	IF State_HS = 0	THEN
		IF SI_MS[0].Event = INIT_CONTINUOUS THEN
			State_MS := 10;
		ELSE
			FSY_In   := FALSE;
			FSY_Out  := FALSE;
			BDef_In  := FALSE;
			BDef_Out := FALSE;
			TDef_In  := FALSE;
			TDef_Out := FALSE;
		END_IF
	END_IF

(*Select MainSail Position*)
10:
	IF END_MS OR Cnt_MS > 10.0 THEN
		State_MS := 0;

	(*1th*)
	ELSIF SI_MS[1].Event = INIT_CONTINUOUS THEN
		Cnt_MS      := 0.0;
		Selected_MS := 1;

		IF TABLE.aFSY [Selected_MS,Selected_HS] = 0
		OR TABLE.aBDef[Selected_MS,Selected_HS] = 0
		OR TABLE.aTDef[Selected_MS,Selected_HS] = 0
		THEN State_MS := 0;
		ELSE State_MS := 11;
		END_IF

	(*2th*)
	ELSIF SI_MS[2].Event = INIT_CONTINUOUS THEN
		Cnt_MS      := 0.0;
		Selected_MS := 2;

		IF TABLE.aFSY [Selected_MS,Selected_HS] = 0
		OR TABLE.aBDef[Selected_MS,Selected_HS] = 0
		OR TABLE.aTDef[Selected_MS,Selected_HS] = 0
		THEN State_MS := 0;
		ELSE State_MS := 12;
		END_IF

	(*3th*)
	ELSIF SI_MS[3].Event = INIT_CONTINUOUS THEN
		Cnt_MS      := 0.0;
		Selected_MS := 3;

		IF TABLE.aFSY [Selected_MS,Selected_HS] = 0
		OR TABLE.aBDef[Selected_MS,Selected_HS] = 0
		OR TABLE.aTDef[Selected_MS,Selected_HS] = 0
		THEN State_MS := 0;
		ELSE State_MS := 13;
		END_IF

	(*FULL*)
	ELSIF SI_MS[4].Event = INIT_CONTINUOUS THEN
		Cnt_MS      := 0.0;
		Selected_MS := 4;

		IF TABLE.aFSY [Selected_MS,Selected_HS] = 0
		OR TABLE.aBDef[Selected_MS,Selected_HS] = 0
		OR TABLE.aTDef[Selected_MS,Selected_HS] = 0
		THEN State_MS := 0;
		ELSE State_MS := 14;
		END_IF

	END_IF

(*Wait 5 Sec*)
11,12,13,14:
	IF END_MS THEN
		State_MS := 0;

	ELSIF Cnt_MS > 5.0 THEN
		Cnt_MS   := 0.0;

		FSY_Tgt := TABLE.aFSY [Selected_MS,Selected_HS];
		FSY_In  := NOT FSY_LS.Err AND FSY_LS.Pos > FSY_Tgt AND NOT FSY_P.AlMax;
		FSY_Out := NOT FSY_LS.Err AND FSY_LS.Pos < FSY_Tgt;

		State_MS := State_MS + 10;

	END_IF

(*Moving Forestay*)
21,22,23,24:
	IF END_MS OR Cnt_MS > 30.0 OR FSY_LS.Err THEN
		State_MS := 0;

	ELSIF FSY_In THEN
		IF FSY_P.AlMax THEN
			State_MS := 0;

		ELSIF FSY_LS.Pos <= FSY_Tgt THEN
			FSY_In   := FALSE;

			BDef_Tgt := TABLE.aBDef[Selected_MS,Selected_HS];
			BDef_In  := NOT BDef_LS.Err AND BDef_LS.Pos > BDef_Tgt AND NOT BDef_P.AlMax;
			BDef_Out := NOT BDef_LS.Err AND BDef_LS.Pos < BDef_Tgt;

			TDef_Tgt := TABLE.aTDef[Selected_MS,Selected_HS];
			TDef_In  := NOT TDef_LS.Err AND TDef_LS.Pos > TDef_Tgt AND NOT TDef_P.AlMax;
			TDef_Out := NOT TDef_LS.Err AND TDef_LS.Pos < TDef_Tgt;

			State_MS := State_MS + 10;

		END_IF

	ELSIF FSY_OUT THEN
		IF FSY_LS.Pos >= FSY_Tgt THEN
			FSY_Out  := FALSE;

			BDef_Tgt := TABLE.aBDef[Selected_MS,Selected_HS];
			BDef_In  := NOT BDef_LS.Err AND BDef_LS.Pos > BDef_Tgt AND NOT BDef_P.AlMax;
			BDef_Out := NOT BDef_LS.Err AND BDef_LS.Pos < BDef_Tgt;

			TDef_Tgt := TABLE.aTDef[Selected_MS,Selected_HS];
			TDef_In  := NOT TDef_LS.Err AND TDef_LS.Pos > TDef_Tgt AND NOT TDef_P.AlMax;
			TDef_Out := NOT TDef_LS.Err AND TDef_LS.Pos < TDef_Tgt;

			State_MS := State_MS + 10;

		END_IF

	ELSE
		State_MS := 0;

	END_IF

(*Moving Deflector*)
31,32,33,34:
	IF END_MS OR Cnt_MS > 30.0 OR BDef_LS.Err OR TDef_LS.Err THEN
		State_MS := 0;

	ELSE
		IF BDef_In THEN
			IF BDef_P.AlMax THEN
				State_MS := 0;
			ELSIF BDef_LS.Pos <= BDef_Tgt THEN
				BDef_In := FALSE;
			END_IF

		ELSIF BDef_Out THEN
			IF BDef_LS.Pos >= BDef_Tgt THEN
				BDef_Out := FALSE;
			END_IF
		END_IF

		IF TDef_In THEN
			IF TDef_P.AlMax THEN
				State_MS := 0;
			ELSIF TDef_LS.Pos <= TDef_Tgt THEN
				TDef_In := FALSE;
			END_IF

		ELSIF TDef_Out THEN
			IF TDef_LS.Pos >= TDef_Tgt THEN
				TDef_Out := FALSE;
			END_IF
		END_IF

		IF NOT BDef_In AND NOT BDef_OUT AND NOT TDef_In AND NOT TDef_Out THEN
			State_MS := 0;
		END_IF

	END_IF

END_CASE

(*HEAD SAIL*)
CASE State_HS OF
0:
	Cnt_HS := 0.0;

	IF State_MS = 0	THEN
		IF SI_HS[0].Event = INIT_CONTINUOUS THEN
			State_HS := 10;
		ELSE
			FSY_In   := FALSE;
			FSY_Out  := FALSE;
			BDef_In  := FALSE;
			BDef_Out := FALSE;
			TDef_In  := FALSE;
			TDef_Out := FALSE;
		END_IF
	END_IF

(*Select HeadSail*)
10:
	IF END_HS OR Cnt_HS > 10.0 THEN
		State_HS := 0;

	(*A3*)
	ELSIF SI_HS[1].Event = INIT_CONTINUOUS THEN
		Cnt_HS      := 0.0;
		Selected_HS := 1;

		IF TABLE.aFSY [Selected_MS,Selected_HS] = 0
		OR TABLE.aBDef[Selected_MS,Selected_HS] = 0
		OR TABLE.aTDef[Selected_MS,Selected_HS] = 0
		THEN State_HS := 0;
		ELSE State_HS := 11;
		END_IF

	(*F0*)
	ELSIF SI_HS[2].Event = INIT_CONTINUOUS THEN
		Cnt_HS      := 0.0;
		Selected_HS := 2;

		IF TABLE.aFSY [Selected_MS,Selected_HS] = 0
		OR TABLE.aBDef[Selected_MS,Selected_HS] = 0
		OR TABLE.aTDef[Selected_MS,Selected_HS] = 0
		THEN State_HS := 0;
		ELSE State_HS := 12;
		END_IF

	(*J2*)
	ELSIF SI_HS[3].Event = INIT_CONTINUOUS THEN
		Cnt_HS      := 0.0;
		Selected_HS := 3;

		IF TABLE.aFSY [Selected_MS,Selected_HS] = 0
		OR TABLE.aBDef[Selected_MS,Selected_HS] = 0
		OR TABLE.aTDef[Selected_MS,Selected_HS] = 0
		THEN State_HS := 0;
		ELSE State_HS := 13;
		END_IF

	(*J4*)
	ELSIF SI_HS[4].Event = INIT_CONTINUOUS THEN
		Cnt_HS      := 0.0;
		Selected_HS := 4;

		IF TABLE.aFSY [Selected_MS,Selected_HS] = 0
		OR TABLE.aBDef[Selected_MS,Selected_HS] = 0
		OR TABLE.aTDef[Selected_MS,Selected_HS] = 0
		THEN State_HS := 0;
		ELSE State_HS := 14;
		END_IF

	END_IF

(*Wait 5 Sec*)
11,12,13,14,15,16:
	IF END_HS THEN
		State_HS := 0;

	(*A3+J4*)
	ELSIF State_HS = 11 AND SI_HS[4].Event = INIT_CONTINUOUS THEN
		Cnt_HS      := 0.0;
		Selected_HS := 5;

		IF TABLE.aFSY [Selected_MS,Selected_HS] = 0
		OR TABLE.aBDef[Selected_MS,Selected_HS] = 0
		OR TABLE.aTDef[Selected_MS,Selected_HS] = 0
		THEN State_HS := 0;
		ELSE State_HS := 15;
		END_IF

	(*F0+J4*)
	ELSIF State_HS = 12 AND SI_HS[4].Event = INIT_CONTINUOUS THEN
		Cnt_HS      := 0.0;
		Selected_HS := 6;

		IF TABLE.aFSY [Selected_MS,Selected_HS] = 0
		OR TABLE.aBDef[Selected_MS,Selected_HS] = 0
		OR TABLE.aTDef[Selected_MS,Selected_HS] = 0
		THEN State_HS := 0;
		ELSE State_HS := 16;
		END_IF

	ELSIF Cnt_HS > 5.0 THEN
		Cnt_HS   := 0.0;

		FSY_Tgt := TABLE.aFSY [Selected_MS,Selected_HS];
		FSY_In  := NOT FSY_LS.Err AND FSY_LS.Pos > FSY_Tgt AND NOT FSY_P.AlMax;
		FSY_Out := NOT FSY_LS.Err AND FSY_LS.Pos < FSY_Tgt;

		State_HS := State_HS + 10;

	END_IF

(*Moving Forestay*)
21,22,23,24,25,26:
	IF END_HS OR Cnt_HS > 30.0 OR FSY_LS.Err THEN
		State_HS := 0;

	ELSIF FSY_In THEN
		IF FSY_P.AlMax THEN
			State_HS := 0;

		ELSIF FSY_LS.Pos <= FSY_Tgt THEN
			FSY_In   := FALSE;

			BDef_Tgt := TABLE.aBDef[Selected_MS,Selected_HS];
			BDef_In  := NOT BDef_LS.Err AND BDef_LS.Pos > BDef_Tgt AND NOT BDef_P.AlMax;
			BDef_Out := NOT BDef_LS.Err AND BDef_LS.Pos < BDef_Tgt;

			TDef_Tgt := TABLE.aTDef[Selected_MS,Selected_HS];
			TDef_In  := NOT TDef_LS.Err AND TDef_LS.Pos > TDef_Tgt AND NOT TDef_P.AlMax;
			TDef_Out := NOT TDef_LS.Err AND TDef_LS.Pos < TDef_Tgt;

			State_HS := State_HS + 10;

		END_IF

	ELSIF FSY_OUT THEN
		IF FSY_LS.Pos >= FSY_Tgt THEN
			FSY_Out  := FALSE;

			BDef_Tgt := TABLE.aBDef[Selected_MS,Selected_HS];
			BDef_In  := NOT BDef_LS.Err AND BDef_LS.Pos > BDef_Tgt AND NOT BDef_P.AlMax;
			BDef_Out := NOT BDef_LS.Err AND BDef_LS.Pos < BDef_Tgt;

			TDef_Tgt := TABLE.aTDef[Selected_MS,Selected_HS];
			TDef_In  := NOT TDef_LS.Err AND TDef_LS.Pos > TDef_Tgt AND NOT TDef_P.AlMax;
			TDef_Out := NOT TDef_LS.Err AND TDef_LS.Pos < TDef_Tgt;

			State_HS := State_HS + 10;

		END_IF

	ELSE
		State_HS := 0;

	END_IF

(*Moving Deflector*)
31,32,33,34,35,36:
	IF END_HS OR Cnt_HS > 30.0 OR BDef_LS.Err OR TDef_LS.Err THEN
		State_HS := 0;

	ELSE
		IF BDef_In THEN
			IF BDef_P.AlMax THEN
				State_HS := 0;
			ELSIF BDef_LS.Pos <= BDef_Tgt THEN
				BDef_In := FALSE;
			END_IF

		ELSIF BDef_Out THEN
			IF BDef_LS.Pos >= BDef_Tgt THEN
				BDef_Out := FALSE;
			END_IF
		END_IF

		IF TDef_In THEN
			IF TDef_P.AlMax THEN
				State_HS := 0;
			ELSIF TDef_LS.Pos <= TDef_Tgt THEN
				TDef_In := FALSE;
			END_IF

		ELSIF TDef_Out THEN
			IF TDef_LS.Pos >= TDef_Tgt THEN
				TDef_Out := FALSE;
			END_IF
		END_IF

		IF NOT BDef_In AND NOT BDef_OUT AND NOT TDef_In AND NOT TDef_Out THEN
			State_HS := 0;
		END_IF

	END_IF

END_CASE
END_FUNCTION_BLOCK

(* POU OUTPUTS, ST *)
PROGRAM OUTPUTS
VAR CONSTANT
	BUF_SIZE : WORD := 4095;
	MAX_PSX  : INT  := 1000; (*100*10*)
END_VAR
VAR
	PSX50 : FB_PSX_VALVE;
	PSX51 : FB_PSX_VALVE;
	PSX52 : FB_PSX_VALVE;
	PSX53 : FB_PSX_VALVE;
	PSX54 : FB_PSX_VALVE;
	PSX55 : FB_PSX_VALVE;
	PSX56 : FB_PSX_VALVE;
	PSX57 : FB_PSX_VALVE;
	PSX58 : FB_PSX_VALVE;
	PSX59 : FB_PSX_VALVE;

	PSX60 : FB_PSX_VALVE;
	PSX61 : FB_PSX_VALVE;
	PSX64 : FB_PSX_VALVE;

	PSX70 : FB_PSX_VALVE;
	PSX71 : FB_PSX_VALVE;
	PSX72 : FB_PSX_VALVE;
	PSX73 : FB_PSX_VALVE;
	PSX74 : FB_PSX_VALVE;

	tsTime    :TIMESTRUCT;
	sDate     :STRING;
	sLocal    :STRING;
	sDaySec   :STRING;


	SIMob      : FB_SMART_INPUT;
	SIDimmerUp : FB_SMART_INPUT;
	SIDimmerDw : FB_SMART_INPUT;

	wDimmerBackLight : WORD;
	byDimmerLedBar   : BYTE;
	byDimmerDeckLink : BYTE;
	byDimmerBLink    : BYTE;
	byDimmerState    : BYTE;

	(*Mob : BOOL;*)

	sValue : STRING;

	engCnt : REAL;

	(*UDP Stream*)
	fbUdpSend        : FB_UDP_SEND;
	fbSocketCloseAll : FB_SocketCloseAll;
    bCloseAll 	     : BOOL := TRUE;

	aBuffer : ARRAY[0..BUF_SIZE] OF BYTE;
	wBufPos : DWORD;

	i   : INT;
	chk : BYTE;
	(*Bobstay_Ignore : BOOL;*)


	fbResetCan1 : IOF_DeviceReset;
	fbResetCan2 : IOF_DeviceReset;
	fbResetCan3 : IOF_DeviceReset;
	fbResetCan4 : IOF_DeviceReset;
	fbResetCan5 : IOF_DeviceReset;

	ResetCan1 : BOOL;
	ResetCan2 : BOOL;
	ResetCan3 : BOOL;
	ResetCan4 : BOOL;
	ResetCan5 : BOOL;

	W_CAN_PWR : BOOL := TRUE;
	W_CAN_CNT : REAL := 20.0;

END_VAR
VAR PERSISTENT
	Dimmer_Panels   AT %Q*: WORD;
	Dimmer_LedBar   AT %Q*: WORD;
	Dimmer_DeckLink AT %Q*: WORD;

END_VAR
W_CAN_CNT := W_CAN_CNT + MAIN.Cycle_Time;
W_CAN_PWR := W_CAN_CNT > 20.0;

(*Node00-PLC*)
N0_DO1 := ALARMS.Buzzer;
(*N0_DO2 := Engine Stop*)
N0_DO3 := W_CAN_PWR;
N0_DO4 := ENGINE.Engine_ON;
(*N0_DO5 := Engine Ignition*)
(*N0_DO6 := Engine Start*)
N0_DO7 := KEY_PP1;
N0_DO8 := KEY_PP2;

N0_AO1 := REAL_TO_INT(THR_PP1 * 3276.7); (*0..10V*)
N0_AO2 := REAL_TO_INT(THR_PP2 * 3276.7); (*0..10V*)


IF NOT TANK.Enable OR ENGINE.Engine_STOP OR NOT MAIN.aSys_Enable[8] THEN

	IF engCnt > 5 THEN
		N0_DO2 := FALSE;
	ELSE
		engCnt := engCnt + MAIN.Cycle_Time;
	END_IF

ELSE
	N0_DO2 := TRUE;


END_IF

(***STERN Nodes***)
(*Node36/37 - TANK + GS + MF00 + PP *)
	N36_EVP3_CH1_2 := EVP001;
	N36_EVP2_CH1_4 := EVP002;

	N36_DO7_CH3_2 := EV1501;
	N36_DO6_CH3_4 := EV1502;

(*Node38 - LIGHT*)
	N38_DO3_CH1_2 := L_Red;
	N38_DO2_CH1_4 := L_Anchor;
	N38_DO1_CH2_2 := L_Steam;
	N38_DO0_CH2_4 := L_Deck;
	N38_DO7_CH3_2 := L_Nav;
(*	N38_DO6_CH3_4 := ;*)
	N38_DO5_CH4_2 := ENGINE.Engine_ON;
	N38_DO4_CH4_4 := ALARMS.Buzzer;

(*Node39 - MF10A - Keel*)
	N39_DO7_CH3_2 := EV1001;
	N39_DO6_CH3_4 := EV1003;
	N39_DO5_CH4_2 := EV1002;
	N39_DO4_CH4_4 := EV1004;

	N39_EVP3_CH1_2 := EVP1006;
	N39_EVP2_CH1_4 := EVP1008;
	N39_EVP1_CH2_2 := EVP1007;
	N39_EVP0_CH2_4 := EVP1009;

(*Node40 - MF10B - Keel*)
	N40_EVP3_CH1_2 := EVP1005.mA := REAL_TO_UINT(EVP1005.Bar * EVP1005.Cal_K + EVP1005.Cal_Off);
	N40_EVP2_CH1_4 := EVP1010.mA := REAL_TO_UINT(EVP1010.Bar * EVP1010.Cal_K + EVP1010.Cal_Off);

	N40_DO1_CH2_2 := EV1011;
	N40_DO0_CH2_4 := EV1012;

(*Node41 - MF05*)
	IF EVP513.Bar > 0 THEN
		N41_EVP3_CH1_2 := EVP513.mA := REAL_TO_UINT(EVP513.Bar * EVP513.Cal_K + EVP513.Cal_Off);
	ELSE
		N41_EVP3_CH1_2 := EVP513.mA := 0;
	END_IF

	N41_DO1_CH2_2 := EV501;
	N41_DO0_CH2_4 := EV502;
	N41_DO7_CH3_2 := EV503;
	N41_DO6_CH3_4 := EV504;
	N41_DO5_CH4_2 := EV505;
	N41_DO4_CH4_4 := EV506;
	N40_DO7_CH3_2 := EV507;
	N40_DO6_CH3_4 := EV508;

(*Node42 - MF01 EVC + PP*)
	N42_DO3_CH1_2 := EV107;
(*	N42_DO2_CH1_4 := *)
	N42_DO1_CH2_2 := EV105;
	N42_DO0_CH2_4 := EV106;
	N42_DO7_CH3_2 := EV103;
	N42_DO6_CH3_4 := EV104;
	N42_DO5_CH4_2 := EV101;
	N42_DO4_CH4_4 := EV102;

(*Node43 - MF03A*)
	N43_DO3_CH1_2 := EV311;
	N43_DO2_CH1_4 := EV312;
	N43_DO1_CH2_2 := EV309;
	N43_DO0_CH2_4 := EV310;
	N43_DO7_CH3_2 := EV307;
	N43_DO6_CH3_4 := EV308;

(*Node44 - MF03A*)
	IF EVP313.Bar > 0 THEN
		N44_EVP3_CH1_2 := EVP313.mA := REAL_TO_UINT(EVP313.Bar * EVP313.Cal_K + EVP313.Cal_Off);
	ELSE
		N44_EVP3_CH1_2 := EVP313.mA := 0;
	END_IF

	N44_DO1_CH2_2 := EV301;
	N44_DO0_CH2_4 := EV302;
	N44_DO7_CH3_2 := EV303;
	N44_DO6_CH3_4 := EV304;
	N44_DO5_CH4_2 := EV305;
	N44_DO4_CH4_4 := EV306;

(*Node48 - DGB Seal*)
	N48_DO3_CH1_2 := EV_SealP_V;
	N48_DO2_CH1_4 := EV_SealP_P;
	N48_DO1_CH2_2 := EV_SealS_V;
	N48_DO0_CH2_4 := EV_SealS_P;

(***STERN Nodes***)
(*Node20 - MF06*)
	N20_DO3_CH1_2 := EV601;
	N20_DO2_CH1_4 := EV602;
	N20_DO1_CH2_2 := EV603;
	N20_DO0_CH2_4 := EV604;
	N20_DO7_CH3_2 := EV605;
	N20_DO6_CH3_4 := EV606;
	N20_DO5_CH4_2 := EV607;
	N20_DO4_CH4_4 := EV608;

(*Node21/22 - MF07 - MF10*)
	IF EVP709.Bar > 0 THEN
		N21_EVP3_CH1_2 := EVP709.mA := REAL_TO_UINT(EVP709.Bar * EVP709.Cal_K + EVP709.Cal_Off);
	ELSE
		N21_EVP3_CH1_2 := EVP709.mA := 0;
	END_IF

	N21_DO1_CH2_2 := EV701;
	N21_DO0_CH2_4 := EV702;
	N21_DO5_CH4_2 := EV703;
	N21_DO4_CH4_4 := EV704;

	N22_DO3_CH1_2 := EV709;
	N22_DO2_CH1_4 := EV710;
	N22_DO1_CH2_2 := EV707;
	N22_DO0_CH2_4 := EV708;
	N22_DO7_CH3_2 := EV705;
	N22_DO6_CH3_4 := EV706;

(*Node23 - MF08*)
	N23_DO3_CH1_2 := EV803;
	N23_DO2_CH1_4 := EV804;
	N23_DO1_CH2_2 := EV801;
	N23_DO0_CH2_4 := EV802;

(*Node26 - MF25*)
	N26_DO3_CH1_2 := EV2502;
	N26_DO2_CH1_4 := EV2504;
	N26_DO1_CH2_2 := EV2501;
	N26_DO0_CH2_4 := EV2503;
	N26_DO7_CH3_2 := EV2506;
	N26_DO6_CH3_4 := EV2508;
	N26_DO5_CH4_2 := EV2505;
	N26_DO4_CH4_4 := EV2507;

(*Node27 - MF22*)
	N27_DO3_CH1_2 := EV2211;
	N27_DO2_CH1_4 := EV2209;
	N27_DO1_CH2_2 := EV2207;
	N27_DO0_CH2_4 := EV2205;
	N27_DO7_CH3_2 := EV2203;
	N27_DO6_CH3_4 := EV2201;

(*Node28 - MF21*)
	N28_DO3_CH1_2 := EV2111;
	N28_DO2_CH1_4 := EV2109;
	N28_DO1_CH2_2 := EV2107;
	N28_DO0_CH2_4 := EV2105;
	N28_DO7_CH3_2 := EV2103;
	N28_DO6_CH3_4 := EV2101;

(*Node29 - MF24*)
	N29_DO3_CH1_2 := EV2411;
	N29_DO2_CH1_4 := EV2409;
	N29_DO1_CH2_2 := EV2407;
	N29_DO0_CH2_4 := EV2405;
	N29_DO7_CH3_2 := EV2403;
	N29_DO6_CH3_4 := EV2401;

(*Node30 - MF23*)
	N30_DO3_CH1_2 := EV2311;
	N30_DO2_CH1_4 := EV2309;
	N30_DO1_CH2_2 := EV2307;
	N30_DO0_CH2_4 := EV2305;
	N30_DO7_CH3_2 := EV2303;
	N30_DO6_CH3_4 := EV2301;

(*Node31 - MF20*)
	N31_DO3_CH1_2 := EV2011;
	N31_DO2_CH1_4 := EV2009;
	N31_DO1_CH2_2 := EV2007;
	N31_DO0_CH2_4 := EV2005;
	N31_DO7_CH3_2 := EV2003;
	N31_DO6_CH3_4 := EV2001;

(*Node32 - MF19*)
	N32_DO3_CH1_2 := EV1911;
	N32_DO2_CH1_4 := EV1909;
	N32_DO1_CH2_2 := EV1907;
	N32_DO0_CH2_4 := EV1905;
	N32_DO7_CH3_2 := EV1903;
	N32_DO6_CH3_4 := EV1901;

(*Node33 - MF13 - Traveller*)
	N33_DO3_CH1_2 := EV1302;
	N33_DO2_CH1_4 := EV1301;
	N33_DO1_CH2_2 := EV1303;

(*Node35 - MF09 - Traveller*)
(*	IF EVP905.Bar > 0 THEN
		N35_EVP3_CH1_2 := EVP905.mA := REAL_TO_UINT(EVP905.Bar * EVP905.Cal_K + EVP905.Cal_Off);
	ELSE
		N35_EVP3_CH1_2 := EVP905.mA := 0;
	END_IF*)

	N35_DO3_CH1_2 := EV905;
	N35_DO2_CH1_4 := EV906;
	N35_DO1_CH2_2 := EV901;
	N35_DO0_CH2_4 := EV902;
	N35_DO7_CH3_2 := EV903;
	N35_DO6_CH3_4 := EV904;
	N35_DO5_CH4_2 := EV907;
	N35_DO4_CH4_4 := EV908;

(*Node47 - MF11*)
	N47_DO1_CH2_2 := EV1101;

(*Node50/59*)
	IF NOT ENGINE.Engine_ON THEN
		IF    EVP402_3 > 0 THEN EVP402_3 :=  MAX_PSX;
		ELSIF EVP402_3 < 0 THEN EVP402_3 := -MAX_PSX;
		END_IF
		IF    EVP404_5 > 0 THEN EVP404_5 :=  MAX_PSX;
		ELSIF EVP404_5 < 0 THEN EVP404_5 := -MAX_PSX;
		END_IF
		IF    EVP406_7 > 0 THEN EVP406_7 :=  MAX_PSX;
		ELSIF EVP406_7 < 0 THEN EVP406_7 := -MAX_PSX;
		END_IF

		IF    EVP1202_3 > 0 THEN EVP1202_3 :=  MAX_PSX;
		ELSIF EVP1202_3 < 0 THEN EVP1202_3 := -MAX_PSX;
		END_IF
		IF    EVP1204_5 > 0 THEN EVP1204_5 :=  MAX_PSX;
		ELSIF EVP1204_5 < 0 THEN EVP1204_5 := -MAX_PSX;
		END_IF
		IF    EVP1206_7 > 0 THEN EVP1206_7 :=  MAX_PSX;
		ELSIF EVP1206_7 < 0 THEN EVP1206_7 := -MAX_PSX;
		END_IF
		IF    EVP1208_9 > 0 THEN EVP1208_9 :=  MAX_PSX;
		ELSIF EVP1208_9 < 0 THEN EVP1208_9 := -MAX_PSX;
		END_IF
		IF    EVP1210_1 > 0 THEN EVP1210_1 :=  MAX_PSX;
		ELSIF EVP1210_1 < 0 THEN EVP1210_1 := -MAX_PSX;
		END_IF
		IF    EVP1212_3 > 0 THEN EVP1212_3 :=  MAX_PSX;
		ELSIF EVP1212_3 < 0 THEN EVP1212_3 := -MAX_PSX;
		END_IF
		IF    EVP1214_5 > 0 THEN EVP1214_5 :=  MAX_PSX;
		ELSIF EVP1214_5 < 0 THEN EVP1214_5 := -MAX_PSX;
		END_IF
		(*IF  EVP1216_7 > 0 THEN EVP1216_7 :=  MAX_PSX; (*Board. Proper value when not Engine.*)
		ELSIF EVP1216_7 < 0 THEN EVP1216_7 := -MAX_PSX;
		END_IF
		IF    EVP1218_9 > 0 THEN EVP1218_9 :=  MAX_PSX;
		ELSIF EVP1218_9 < 0 THEN EVP1218_9 := -MAX_PSX;
		END_IF*)
		(*IF  EVP1220_1 > 0 THEN EVP1220_1 :=  MAX_PSX; (*Keel Fill. Not Without Engine.*)
		ELSIF EVP1220_1 < 0 THEN EVP1220_1 :=  0;
		END_IF*)

		IF    EVP1602_3 > 0 THEN EVP1602_3 :=  MAX_PSX;
		ELSIF EVP1602_3 < 0 THEN EVP1602_3 := -MAX_PSX;
		END_IF
		IF    EVP1604_5 > 0 THEN EVP1604_5 :=  MAX_PSX;
		ELSIF EVP1604_5 < 0 THEN EVP1604_5 := -MAX_PSX;
		END_IF
		IF    EVP1606_7 > 0 THEN EVP1606_7 :=  MAX_PSX;
		ELSIF EVP1606_7 < 0 THEN EVP1606_7 := -MAX_PSX;
		END_IF
		IF    EVP1608_9 > 0 THEN EVP1608_9 :=  MAX_PSX;
		ELSIF EVP1608_9 < 0 THEN EVP1608_9 := -MAX_PSX;
		END_IF
		IF    EVP1610_1 > 0 THEN EVP1610_1 :=  MAX_PSX;
		ELSIF EVP1610_1 < 0 THEN EVP1610_1 := -MAX_PSX;
		END_IF

	END_IF

	PSX50( SP:= EVP1202_3, IN:= N50_IN, OUT:= N50_OUT );
	PSX51( SP:= EVP1204_5, IN:= N51_IN, OUT:= N51_OUT );
	PSX52( SP:= EVP1206_7, IN:= N52_IN, OUT:= N52_OUT );
	PSX53( SP:= EVP1208_9, IN:= N53_IN, OUT:= N53_OUT );
	PSX54( SP:= EVP1210_1, IN:= N54_IN, OUT:= N54_OUT );
	PSX55( SP:= EVP1212_3, IN:= N55_IN, OUT:= N55_OUT );
	PSX56( SP:= EVP1214_5, IN:= N56_IN, OUT:= N56_OUT );
	PSX57( SP:= EVP1216_7, IN:= N57_IN, OUT:= N57_OUT );
	PSX58( SP:= EVP1218_9, IN:= N58_IN, OUT:= N58_OUT );
	PSX59( SP:= EVP1220_1, IN:= N59_IN, OUT:= N59_OUT );

	PSX60( SP:= EVP402_3, IN:= N60_IN, OUT:= N60_OUT );
	PSX61( SP:= EVP404_5, IN:= N61_IN, OUT:= N61_OUT );
	PSX64( SP:= EVP406_7, IN:= N64_IN, OUT:= N64_OUT );

	PSX70( SP:= EVP1602_3, IN:= N70_IN, OUT:= N70_OUT );
	PSX71( SP:= EVP1604_5, IN:= N71_IN, OUT:= N71_OUT );
	PSX72( SP:= EVP1606_7, IN:= N72_IN, OUT:= N72_OUT );
	PSX73( SP:= EVP1608_9, IN:= N73_IN, OUT:= N73_OUT );
	PSX74( SP:= EVP1610_1, IN:= N74_IN, OUT:= N74_OUT );

(*-------------------*)
(*-- Panel Buttons --*)
(*-------------------*)
SIDimmerUp( T_Cont:= T#0ms, T_DClk:= T#0ms);
SIDimmerDw(In:= N103_IN.5, T_Cont:= T#0ms, T_DClk:= T#0ms);

IF SIDimmerUp.Event = INIT_CONTINUOUS
OR SIDimmerDw.Event = INIT_CONTINUOUS
THEN

	IF byDimmerState = 2
	THEN byDimmerState := 0;
	ELSE byDimmerState := byDimmerState + 1;
	END_IF

END_IF

CASE byDimmerState OF
0:
	wDimmerBackLight := 100;
	byDimmerLedBar   := 16#9F; (*16#80 + 16#1F*)
	byDimmerDeckLink := 16#07;
	byDimmerBLink    := 16#3F;

1:
	wDimmerBackLight := Dimmer_Panels;
	byDimmerLedBar   := REAL_TO_USINT(Dimmer_LedBar   * 0.31) + 16#80;
	byDimmerDeckLink := REAL_TO_USINT(Dimmer_DEckLink * 0.07);
	byDimmerBLink    := REAL_TO_USINT(Dimmer_Panels   * 0.63);

2:
	wDimmerBackLight := 100;
	byDimmerLedBar   := 16#9F; (*16#80 + 16#1F*)
	byDimmerDeckLink := 16#07;
	byDimmerBLink    := 16#3F;

END_CASE

IF byDimmerState > 0 AND MAIN.aSys_Enable[2] AND wDimmerBackLight > 0 THEN
	N102_OUT := 16#FFFF;
	N103_OUT := 16#FFFF;
	N104_OUT := 16#FFFF;
	N105_OUT := 16#FFFF;
	N106_OUT := 16#FFFF;
	N107_OUT := 16#FFFF;
	N108_OUT := 16#FFE0;
	N109_OUT := 16#FFE0;
	N110_OUT := 16#FFFF;
	N111_OUT := 16#FFFF;
	N112_OUT := 16#FFFF;
	N113_OUT := 16#FFFF;
	N114_OUT := 16#FFFF;
	N115_OUT := 16#FFFF;
	N116_OUT := 16#FFFF;
	N117_OUT := 16#FFFF;
	N118_OUT := 16#FFFF;
	N119_OUT := 16#FFFF;

	N120_LED_R := 16#0000;
	N120_LED_G := 16#03DE;
	N120_LED_B := 16#0021;
	N121_LED_R := 16#00FF;
	N121_LED_G := 16#0000;
	N121_LED_B := 16#0000;

ELSE
	N102_OUT := 0;
	N103_OUT := 0;
	N104_OUT := 0;
	N105_OUT := 0;
	N106_OUT := 0;
	N107_OUT := 0;
	N108_OUT := 0;
	N109_OUT := 0;
	N110_OUT := 0;
	N111_OUT := 0;
	N112_OUT := 0;
	N113_OUT := 0;
	N114_OUT := 0;
	N115_OUT := 0;
	N116_OUT := 0;
	N117_OUT := 0;
	N118_OUT := 0;
	N119_OUT := 0;

	N120_LED_R := 0;
	N120_LED_G := 0;
	N120_LED_B := 0;
	N121_LED_R := 0;
	N121_LED_G := 0;
	N121_LED_B := 0;
END_IF

IF wDimmerBackLight = 0 THEN wDimmerBackLight := 1; END_IF

N102_DIMMER := wDimmerBackLight;
N103_DIMMER := wDimmerBackLight;
N104_DIMMER := wDimmerBackLight;
N105_DIMMER := wDimmerBackLight;
N106_DIMMER := wDimmerBackLight;
N107_DIMMER := wDimmerBackLight;
N108_DIMMER := wDimmerBackLight;
N109_DIMMER := wDimmerBackLight;
N110_DIMMER := wDimmerBackLight;
N111_DIMMER := wDimmerBackLight;
N112_DIMMER := wDimmerBackLight;
N113_DIMMER := wDimmerBackLight;
N114_DIMMER := wDimmerBackLight;
N115_DIMMER := wDimmerBackLight;
N116_DIMMER := wDimmerBackLight;
N117_DIMMER := wDimmerBackLight;
N118_DIMMER := wDimmerBackLight;
N119_DIMMER := wDimmerBackLight;

N120_LED_Bright := byDimmerBLink;
N121_LED_Bright := byDimmerBLink;

N102_BTIME := 10;
N103_BTIME := 10;
N104_BTIME := 10;
N105_BTIME := 10;
IF MAIN.fbWB.Pause THEN
	N106_BTIME := 100;
	N107_BTIME := 100;
ELSE
	N106_BTIME := 10;
	N107_BTIME := 10;
END_IF
N108_BTIME := 10;
N109_BTIME := 10;
N110_BTIME := 10;
N111_BTIME := 10;
N112_BTIME := 10;
N113_BTIME := 10;
N114_BTIME := 10;
N115_BTIME := 10;
N116_BTIME := 10;
N117_BTIME := 10;
N118_BTIME := 10;
N119_BTIME := 10;

(*FRO TACK*)
N102_BLINK.2 := MAIN.fbSE301.OUT_CylIn;
N102_BLINK.3 := MAIN.fbSE301.OUT_CylOut;
N113_BLINK.3 := MAIN.fbSE301.OUT_CylIn;
N113_BLINK.2 := MAIN.fbSE301.OUT_CylOut;
(*A3 TACK*)
N102_BLINK.4 := MAIN.fbSE303.OUT_CylIn;
N102_BLINK.5 := MAIN.fbSE303.OUT_CylOut;
N113_BLINK.5 := MAIN.fbSE303.OUT_CylIn;
N113_BLINK.4 := MAIN.fbSE303.OUT_CylOut;
(*J5*)
N118_BLINK.6 := MAIN.fbSE305.OUT_CylIn;
N118_BLINK.7 := MAIN.fbSE305.OUT_CylOut;
N119_BLINK.7 := MAIN.fbSE305.OUT_CylIn;
N119_BLINK.6 := MAIN.fbSE305.OUT_CylOut;
(*J4*)
N118_BLINK.8 := MAIN.fbSE307.OUT_CylIn;
N118_BLINK.9 := MAIN.fbSE307.OUT_CylOut;
N119_BLINK.9 := MAIN.fbSE307.OUT_CylIn;
N119_BLINK.8 := MAIN.fbSE307.OUT_CylOut;
(*FORESTAY*)
N104_BLINK.1 := MAIN.fbSE309.OUT_CylIn;
N104_BLINK.0 := MAIN.fbSE309.OUT_CylOut;
N105_BLINK.0 := MAIN.fbSE309.OUT_CylIn;
N105_BLINK.1 := MAIN.fbSE309.OUT_CylOut;
(*J2*)
N114_BLINK.4 := MAIN.fbSE311.OUT_CylIn;
N114_BLINK.5 := MAIN.fbSE311.OUT_CylOut;
N115_BLINK.5 := MAIN.fbSE311.OUT_CylIn;
N115_BLINK.4 := MAIN.fbSE311.OUT_CylOut;

(*JIB INOUT*)
N114_BLINK.2 := MAIN.fbSE501.OUT_CylIn;
N114_BLINK.3 := MAIN.fbSE501.OUT_CylOut;
N115_BLINK.3 := MAIN.fbSE501.OUT_CylIn;
N115_BLINK.2 := MAIN.fbSE501.OUT_CylOut;
(*JIB UPDW*)
N114_BLINK.0 := MAIN.fbSE503.OUT_CylIn;
N114_BLINK.1 := MAIN.fbSE503.OUT_CylOut;
N115_BLINK.1 := MAIN.fbSE503.OUT_CylIn;
N115_BLINK.0 := MAIN.fbSE503.OUT_CylOut;
(*VANG*)
N116_BLINK.2 := MAIN.fbSE505.OUT_CylIn;
N116_BLINK.3 := MAIN.fbSE505.OUT_CylOut;
N117_BLINK.3 := MAIN.fbSE505.OUT_CylIn;
N117_BLINK.2 := MAIN.fbSE505.OUT_CylOut;

(*PROP UPDW*)
N112_BLINK.3 := MAIN.fbDE601.OUT_EV3;
N112_BLINK.2 := MAIN.fbDE601.OUT_EV1;
(*TRIM TAB*)
N104_BLINK.3 := MAIN.fbDE605.OUT_EV3;
N104_BLINK.2 := MAIN.fbDE605.OUT_EV1;
N105_BLINK.3 := MAIN.fbDE605.OUT_EV3;
N105_BLINK.2 := MAIN.fbDE605.OUT_EV1;

(*INNER STAYSAIL*)
N102_BLINK.0 := MAIN.fbSE701.OUT_CylIn;
N102_BLINK.1 := MAIN.fbSE701.OUT_CylOut;
N113_BLINK.1 := MAIN.fbSE701.OUT_CylIn;
N113_BLINK.0 := MAIN.fbSE701.OUT_CylOut;
(*MAIN OUTHAUL*)
N116_BLINK.8 := MAIN.fbSE703.OUT_CylIn;
N116_BLINK.9 := MAIN.fbSE703.OUT_CylOut;
N117_BLINK.9 := MAIN.fbSE703.OUT_CylIn;
N117_BLINK.8 := MAIN.fbSE703.OUT_CylOut;
(*MAIN CUNN*)
N116_BLINK.6 := MAIN.fbSE705.OUT_CylIn;
N116_BLINK.7 := MAIN.fbSE705.OUT_CylOut;
N117_BLINK.7 := MAIN.fbSE705.OUT_CylIn;
N117_BLINK.6 := MAIN.fbSE705.OUT_CylOut;
(*BOTTOM DEF*)
N118_BLINK.2 := MAIN.fbSE707.OUT_CylIn;
N118_BLINK.3 := MAIN.fbSE707.OUT_CylOut;
N119_BLINK.3 := MAIN.fbSE707.OUT_CylIn;
N119_BLINK.2 := MAIN.fbSE707.OUT_CylOut;
(*BOTTOM DEF*)
N118_BLINK.4 := MAIN.fbSE709.OUT_CylIn;
N118_BLINK.5 := MAIN.fbSE709.OUT_CylOut;
N119_BLINK.5 := MAIN.fbSE709.OUT_CylIn;
N119_BLINK.4 := MAIN.fbSE709.OUT_CylOut;

(*BACKSTAY PORT*)
N104_BLINK.7 := MAIN.fbBSY.OUT_P_In;
N104_BLINK.6 := MAIN.fbBSY.OUT_P_Out;
N118_BLINK.0 := MAIN.fbBSY.OUT_P_In;
N118_BLINK.1 := MAIN.fbBSY.OUT_P_Out;
(*BACKSTAY STBD*)
N105_BLINK.6 := MAIN.fbBSY.OUT_S_In;
N105_BLINK.7 := MAIN.fbBSY.OUT_S_Out;
N119_BLINK.1 := MAIN.fbBSY.OUT_S_In;
N119_BLINK.0 := MAIN.fbBSY.OUT_S_Out;
(*BACKSTAY TACK*)
(*N104_BLINK.5 :=;*)
(*N105_BLINK.4 :=;*)

(*TRAVELLER*)
N116_BLINK.3 := MAIN.fbTraveller.Move_A;
N116_BLINK.2 := MAIN.fbTraveller.Move_B;
(*N116_BLINK.1 := ;*)
N116_BLINK.0 := MAIN.fbTraveller.OUT_EVAB;

N117_BLINK.3 := MAIN.fbTraveller.Move_A;
N117_BLINK.2 := MAIN.fbTraveller.Move_B;
(*N117_BLINK.0 := ;*)
N117_BLINK.1 := MAIN.fbTraveller.OUT_EVAB;

(*KEEL*)
N110_BLINK.0 := MAIN.fbKeel.MOVING_O;
N110_BLINK.4 := MAIN.fbKeel.MOVING_I;
N110_BLINK.3 := MAIN.fbKeel.MOVING_C;
N110_BLINK.2 := MAIN.fbKeel.MOVING_F;
N110_BLINK.5 := MAIN.fbKeel.MOVING_T;

N111_BLINK.0 := MAIN.fbKeel.MOVING_O;
N111_BLINK.4 := MAIN.fbKeel.MOVING_I;
N111_BLINK.3 := MAIN.fbKeel.MOVING_C;
N111_BLINK.2 := MAIN.fbKeel.MOVING_F;
N111_BLINK.5 := MAIN.fbKeel.MOVING_T;

(*N108_BLINK.0 := MAIN.fbKeel.MOVING_O;
N108_BLINK.4 := MAIN.fbKeel.MOVING_I;
N108_BLINK.3 := MAIN.fbKeel.MOVING_C;
N108_BLINK.2 := MAIN.fbKeel.MOVING_F;

N109_BLINK.0 := MAIN.fbKeel.MOVING_O;
N109_BLINK.4 := MAIN.fbKeel.MOVING_I;
N109_BLINK.3 := MAIN.fbKeel.MOVING_C;
N109_BLINK.2 := MAIN.fbKeel.MOVING_F;*) (*Now Mast setup*)

(*WINCHES*)
N117_BLINK.1 := INPUTS.Override_ON;
N105_BLINK.4 := INPUTS.RemPort_ON;
N104_BLINK.5 := INPUTS.RemStbd_ON;

(*MAINSAIL*)
CASE MAIN.fbMastSetup.State_MS OF
0: 	N109_BLINK.0 := N109_BLINK.4 := N109_BLINK.3 := N109_BLINK.2 := FALSE;

10:	N109_BLINK.0 := N109_BLINK.4 := N109_BLINK.3 := N109_BLINK.2 := TRUE;

11: N109_OUT.2   := TRUE;
	N109_BLINK.0 := N109_BLINK.4 := N109_BLINK.3 := N109_BLINK.2 := FALSE;

12: N109_OUT.4   := TRUE;
	N109_BLINK.0 := N109_BLINK.4 := N109_BLINK.3 := N109_BLINK.2 := FALSE;

13: N109_OUT.3   := TRUE;
	N109_BLINK.0 := N109_BLINK.4 := N109_BLINK.3 := N109_BLINK.2 := FALSE;

14: N109_OUT.0   := TRUE;
	N109_BLINK.0 := N109_BLINK.4 := N109_BLINK.3 := N109_BLINK.2 := FALSE;

21,31:
	N109_BLINK.2 := TRUE;
	N109_BLINK.0 := N109_BLINK.4 := N109_BLINK.3 := FALSE;

22,32:
	N109_BLINK.4 := TRUE;
	N109_BLINK.0 := N109_BLINK.3 := N109_BLINK.2 := FALSE;

23,33:
	N109_BLINK.3 := TRUE;
	N109_BLINK.0 := N109_BLINK.4 := N109_BLINK.2 := FALSE;

24,34:
	N109_BLINK.0 := TRUE;
	N109_BLINK.4 := N109_BLINK.3 := N109_BLINK.2 := FALSE;

END_CASE

(*HEADSAIL*)
CASE MAIN.fbMastSetup.State_HS OF
0: 	N108_BLINK.0 := N108_BLINK.4 := N108_BLINK.3 := N108_BLINK.2 := FALSE;

10: N108_BLINK.0 := N108_BLINK.4 := N108_BLINK.3 := N108_BLINK.2 := TRUE;

11:	N108_OUT.0   := TRUE;
	N108_BLINK.0 := N108_BLINK.4 := N108_BLINK.3 := N108_BLINK.2 := FALSE;

12:	N108_OUT.4   := TRUE;
	N108_BLINK.0 := N108_BLINK.4 := N108_BLINK.3 := N108_BLINK.2 := FALSE;

13:	N108_OUT.2   := TRUE;
	N108_BLINK.0 := N108_BLINK.4 := N108_BLINK.3 := N108_BLINK.2 := FALSE;

14:	N108_OUT.3   := TRUE;
	N108_BLINK.0 := N108_BLINK.4 := N108_BLINK.3 := N108_BLINK.2 := FALSE;

15:	N108_OUT.0   := N108_OUT.3   := TRUE;
	N108_BLINK.0 := N108_BLINK.4 := N108_BLINK.3 := N108_BLINK.2 := FALSE;

16:	N108_OUT.4   := N108_OUT.3   := TRUE;
	N108_BLINK.0 := N108_BLINK.4 := N108_BLINK.3 := N108_BLINK.2 := FALSE;

21,31:
	N108_BLINK.0 := TRUE;
	N108_BLINK.4 := N108_BLINK.3 := N108_BLINK.2 := FALSE;

22,32:
	N108_BLINK.4 := TRUE;
	N108_BLINK.0 := N108_BLINK.3 := N108_BLINK.2 := FALSE;

23,33:
	N108_BLINK.2 := TRUE;
	N108_BLINK.0 := N108_BLINK.4 := N108_BLINK.3 := FALSE;

24,34:
	N108_BLINK.3 := TRUE;
	N108_BLINK.0 := N108_BLINK.4 := N108_BLINK.2 := FALSE;

25,35:
	N108_BLINK.0 := N108_BLINK.3 := TRUE;
	N108_BLINK.4 := N108_BLINK.2 := FALSE;

26,36:
	N108_BLINK.4 := N108_BLINK.3 := TRUE;
	N108_BLINK.0 := N108_BLINK.2 := FALSE;

END_CASE

(*BOARD*)
N108_BLINK.6 := MAIN.fbBoard.MOVING_P;
N108_BLINK.7 := MAIN.fbBoard.MOVING_S;
N108_BLINK.5 := MAIN.fbBoard.MOVING_C;

N109_BLINK.6 := MAIN.fbBoard.MOVING_P;
N109_BLINK.7 := MAIN.fbBoard.MOVING_S;
N109_BLINK.5 := MAIN.fbBoard.MOVING_C;

(*BOW THR*)
N112_BLINK.4 := MAIN.fbBowThrUpDw.OUT_1;
N112_BLINK.5 := MAIN.fbBowThrUpDw.OUT_2;

(*Water Ballast*)
N106_BLINK.0 := N107_BLINK.0 := MAIN.fbWB.OUT_P_Fwd;
N106_BLINK.1 := N107_BLINK.1 := MAIN.fbWB.OUT_S_Fwd;
N106_BLINK.2 := N107_BLINK.2 := MAIN.fbWB.OUT_P_Aft;
N106_BLINK.3 := N107_BLINK.3 := MAIN.fbWB.OUT_S_Aft;
N106_BLINK.4 := N107_BLINK.4 := MAIN.fbWB.OUT_Fill;
N106_BLINK.5 := N107_BLINK.5 := MAIN.fbWB.OUT_Dump;
N106_BLINK.7 := N107_BLINK.7 := MAIN.fbWB.OUT_Stop;
N106_BLINK.8 := N107_BLINK.8 := MAIN.fbWB.OUT_12;
N106_BLINK.9 := N107_BLINK.9 := MAIN.fbWB.OUT_Move;

N120_BLINK_B.0 := MAIN.fbW1206.Out_1;
N120_BLINK_G.1 := MAIN.fbW1204.Out_1;
N120_BLINK_G.2 := MAIN.fbW1604.Out_1;
N120_BLINK_G.3 := MAIN.fbW1202.Out_1;
N120_BLINK_G.4 := MAIN.fbW1602.Out_1;
N120_BLINK_B.5 := MAIN.fbW1206.Out_2;
N120_BLINK_G.6 := MAIN.fbW1204.Out_2;
N120_BLINK_G.7 := MAIN.fbW1604.Out_2;
N120_BLINK_G.8 := MAIN.fbW1202.Out_2;
N120_BLINK_G.9 := MAIN.fbW1602.Out_2;

N121_BLINK_R.0 := MAIN.fbW1208.Out_1;
N121_BLINK_R.1 := MAIN.fbW1210.Out_1;
N121_BLINK_R.2 := MAIN.fbW1212.Out_1;
N121_BLINK_R.3 := MAIN.fbW1214.Out_1;
N121_BLINK_R.4 := MAIN.fbW1208.Out_2;
N121_BLINK_R.5 := MAIN.fbW1210.Out_2;
N121_BLINK_R.6 := MAIN.fbW1212.Out_2;
N121_BLINK_R.7 := MAIN.fbW1214.Out_2;

(*CLM8*)
CLM8_LED1.7 := TOFARO.rBar1 >= 100;
CLM8_LED1.6 := TOFARO.rBar1 >= 95;
CLM8_LED1.5 := TOFARO.rBar1 >= 90;
CLM8_LED1.4 := TOFARO.rBar1 >= 85;
CLM8_LED1.3 := TOFARO.rBar1 >= 68;
CLM8_LED1.2 := TOFARO.rBar1 >= 51;
CLM8_LED1.1 := TOFARO.rBar1 >= 34;
CLM8_LED1.0 := TOFARO.rBar1 >= 17;

CLM8_LED2.0 := TOFARO.rBar2 >= 100;
CLM8_LED2.1 := TOFARO.rBar2 >= 95;
CLM8_LED2.2 := TOFARO.rBar2 >= 90;
CLM8_LED2.3 := TOFARO.rBar2 >= 85;
CLM8_LED2.4 := TOFARO.rBar2 >= 68;
CLM8_LED2.5 := TOFARO.rBar2 >= 51;
CLM8_LED2.6 := TOFARO.rBar2 >= 34;
CLM8_LED2.7 := TOFARO.rBar2 >= 17;

IF TOFARO.rBar1 >= 105 THEN
				   (*7888____5556667722333444____1112*)
				   (*RBGR____BGRBGRBGGRBGRBGR____BGRB*)
	CLM8_COLOR1 := 2#10010000001001000100100100000010;
ELSE
				   (*7888____5556667722333444____1112*)
				   (*RBGR____BGRBGRBGGRBGRBGR____BGRB*)
	CLM8_COLOR1 := 2#10010000011011001001001000000100;
END_IF

IF TOFARO.rBar2 >= 105 THEN
				   (*7888____5556667722333444____1112*)
				   (*RBGR____BGRBGRBGGRBGRBGR____BGRB*)
	CLM8_COLOR2 := 2#10010000001001000100100100000010;
ELSE
				   (*7888____5556667722333444____1112*)
				   (*RBGR____BGRBGRBGGRBGRBGR____BGRB*)
	CLM8_COLOR2 := 2#00100000010010010101101100000010;
END_IF

CLM8_BRIGHT := byDimmerLedBar;

(*DeckLink*)
(*N02_OUT.0 := MAIN.aSys_Enable[2];
N03_OUT.0 := MAIN.aSys_Enable[2];
N04_OUT.0 := MAIN.aSys_Enable[2];
N05_OUT.0 := MAIN.aSys_Enable[2];
N06_OUT.0 := MAIN.aSys_Enable[2];
N07_OUT.0 := MAIN.aSys_Enable[2];
N08_OUT.0 := MAIN.aSys_Enable[2];
N09_OUT.0 := MAIN.aSys_Enable[2];
N10_OUT.0 := MAIN.aSys_Enable[2];
N11_OUT.0 := MAIN.aSys_Enable[2];
N12_OUT.0 := MAIN.aSys_Enable[2];
N13_OUT.0 := MAIN.aSys_Enable[2];
N14_OUT.0 := MAIN.aSys_Enable[2];
N15_OUT.0 := MAIN.aSys_Enable[2];
N16_OUT.0 := MAIN.aSys_Enable[2];
N17_OUT.0 := MAIN.aSys_Enable[2];
N18_OUT.0 := MAIN.aSys_Enable[2];
N19_OUT.0 := MAIN.aSys_Enable[2];
N20_OUT.0 := MAIN.aSys_Enable[2];
N21_OUT.0 := MAIN.aSys_Enable[2];

N02_DIMMER := byDimmerDeckLink;
N03_DIMMER := byDimmerDeckLink;
N04_DIMMER := byDimmerDeckLink;
N05_DIMMER := byDimmerDeckLink;
N06_DIMMER := byDimmerDeckLink;
N07_DIMMER := byDimmerDeckLink;
N08_DIMMER := byDimmerDeckLink;
N09_DIMMER := byDimmerDeckLink;
N10_DIMMER := byDimmerDeckLink;
N11_DIMMER := byDimmerDeckLink;
N12_DIMMER := byDimmerDeckLink;
N13_DIMMER := byDimmerDeckLink;
N14_DIMMER := byDimmerDeckLink;
N15_DIMMER := byDimmerDeckLink;
N16_DIMMER := byDimmerDeckLink;
N17_DIMMER := byDimmerDeckLink;
N18_DIMMER := byDimmerDeckLink;
N19_DIMMER := byDimmerDeckLink;
N20_DIMMER := byDimmerDeckLink;
N21_DIMMER := byDimmerDeckLink;

(*Main*)                  (*_LPI*)
N02_COLOR := N03_COLOR:= 16#0203;
N21_COLOR := N20_COLOR:= 16#0203;

(*Port*)                  (*_LPI*)
N04_COLOR := N05_COLOR:= 16#0011;
N08_COLOR := N09_COLOR:= 16#0011;
N14_COLOR := N15_COLOR:= 16#0011;
N18_COLOR := N19_COLOR:= 16#0011;

(*Stbd*)                  (*_LPI*)
N06_COLOR := N07_COLOR:= 16#0122;
N10_COLOR := N11_COLOR:= 16#0122;
N12_COLOR := N13_COLOR:= 16#0122;
N16_COLOR := N17_COLOR:= 16#0122;

(*Primary Stbd/Port*)
IF    INPUTS.C_PS THEN N14_COLOR := N15_COLOR:= 16#0122; (*_LPI*)
ELSIF INPUTS.C_PP THEN N12_COLOR := N13_COLOR:= 16#0011; (*_LPI*)
END_IF

(*Sec. Stbd/Port*)
IF    INPUTS.C_SS THEN N18_COLOR := N19_COLOR:= 16#0122; (*_LPI*)
ELSIF INPUTS.C_SP THEN N16_COLOR := N17_COLOR:= 16#0011; (*_LPI*)
END_IF

(*Main*)
IF    INPUTS.C_MP1 THEN N14_COLOR := N15_COLOR := 16#0203; (*_LPI*)
ELSIF INPUTS.C_MP2 THEN N04_COLOR := N05_COLOR := 16#0203; (*_LPI*)
ELSIF INPUTS.C_MS1 THEN N12_COLOR := N13_COLOR := 16#0203; (*_LPI*)
ELSIF INPUTS.C_MS2 THEN N06_COLOR := N07_COLOR := 16#0203; (*_LPI*)
END_IF**)

(*Reset CAN BUS*)
fbResetCan1 ( DEVICEID:=  2, RESET:= ResetCan1, TMOUT:= T#20s );
fbResetCan2 ( DEVICEID:=  3, RESET:= ResetCan2, TMOUT:= T#20s );
fbResetCan3 ( DEVICEID:=  4, RESET:= ResetCan3, TMOUT:= T#20s );
fbResetCan4 ( DEVICEID:=  5, RESET:= ResetCan4, TMOUT:= T#20s );
fbResetCan5 ( DEVICEID:=  7, RESET:= ResetCan5, TMOUT:= T#20s );

IF ResetCan1 THEN ResetCan1 := FALSE; END_IF
IF ResetCan2 THEN ResetCan2 := FALSE; END_IF
IF ResetCan3 THEN ResetCan3 := FALSE; END_IF
IF ResetCan4 THEN ResetCan4 := FALSE; END_IF
IF ResetCan5 THEN ResetCan5 := FALSE; END_IF
END_PROGRAM

(* POU FB/FB_PSX_VALVE, ST *)
FUNCTION_BLOCK FB_PSX_VALVE
VAR_INPUT
	SP : INT;
END_VAR
VAR_IN_OUT
	IN  : ST_PSX_VALVE_IN;
	OUT : ST_PSX_VALVE_OUT;
END_VAR
VAR_OUTPUT
END_VAR
VAR
	State : WORD;

END_VAR
(*
  CONTROL				STATUS
0 Disable 				Disabled
1 Hold Enable 			Hold Enabled
2 Device Mode Active 	Device Mode Active
3 Reset Fault 			Ready
14 Second Ramp Set
15 floating position
*)
(* ERROR

0 Internal error (Selftest)
1 Error Buscommand (Timeout, SP value)
2 Coil ressitance, current control
3 Overheating, limited functionallity
4 Spool position too far out
5 Spool position can NOT reach target
6 Setpoint after restart != 0
7 Supply voltage too high/low
8 Temperature too low
9 Temperature too high
10 Parameter/Valve data invalid
11 Sticky spool movement
12 -
13 -
14 Position detectiuon failure
15 Status message, System alive
*)
CASE IN.Status OF

16#01:
	IF IN.Error = 16#8000 THEN
		OUT.Control  := 16#01;
		OUT.SetPoint := 16#00;
	ELSE
		OUT.Control  := 16#08;
		OUT.SetPoint := 16#00;
	END_IF

16#09:
	OUT.Control  := 16#07;
	OUT.SetPoint := 16#00;

16#0F:
	OUT.Control  := 16#07;
	OUT.SetPoint := SP;

ELSE
	IF IN.Error = 16#8000 THEN
		OUT.Control  := 16#01;
		OUT.SetPoint := 16#00;
	ELSE
		OUT.Control  := 16#08;
		OUT.SetPoint := 16#00;
	END_IF

END_CASE
END_FUNCTION_BLOCK

(* POU J1939, ST *)
PROGRAM J1939
VAR CONSTANT
	Cycle_Time1 : REAL := 0.005; (*5ms*)
END_VAR
VAR
END_VAR
PARAMS; (*To Load Faster*)

(**********)
(* ENGINE *)
(**********)
RECV_J1939;
SEND_J1939;
END_PROGRAM

(* POU FB/CobIdDataVisualize, ST *)
FUNCTION_BLOCK CobIdDataVisualize
VAR_INPUT
	rxData : POINTER TO ARRAY [0..7] OF USINT;
END_VAR
VAR_OUTPUT
	strRxData:STRING;
END_VAR
VAR
	f0 : FB_FormatString;
END_VAR
f0(
	sFormat:='%0.2X %0.2X %0.2X %0.2X %0.2X %0.2X %0.2X %0.2X ' ,
	arg1:=F_USINT(rxData^[0]),
	arg2:=F_USINT(rxData^[1]) ,
	arg3:=F_USINT(rxData^[2]) ,
	arg4:= F_USINT(rxData^[3]),
	arg5:=F_USINT(rxData^[4]) ,
	arg6:= F_USINT(rxData^[5]),
	arg7:=F_USINT(rxData^[6]) ,
	arg8:= F_USINT(rxData^[7]),
	arg9:= , 
	arg10:= , 
	bError=> , 
	nErrId=> , 
	sOut=>strRxData );
END_FUNCTION_BLOCK

(* POU FUN/PARAMETERS/F_READ_LIFT_KEEL_CFG, ST *)
FUNCTION F_READ_LIFT_KEEL_CFG : BOOL
VAR_INPUT
	sHead : STRING;
	rTime : REAL;
END_VAR
VAR_IN_OUT
	stConfig : ST_LIFT_KEEL_CFG;
	fbIdList : FB_IDLIST;
END_VAR
VAR
END_VAR
stConfig.PMax_Up := F_IDLIST_GETREAL( CONCAT(sHead, '_PMax_Up' ), fbIdList );
stConfig.PMax_Dw := F_IDLIST_GETREAL( CONCAT(sHead, '_PMax_Dw' ), fbIdList );
stConfig.P500_Up := F_IDLIST_GETREAL( CONCAT(sHead, '_P500_Up' ), fbIdList );
stConfig.P500_Dw := F_IDLIST_GETREAL( CONCAT(sHead, '_P500_Dw' ), fbIdList );
stConfig.P144_F  := F_IDLIST_GETREAL( CONCAT(sHead, '_P144_F'  ), fbIdList );
stConfig.P144_S  := F_IDLIST_GETREAL( CONCAT(sHead, '_P144_S'  ), fbIdList );

stConfig.TgtP_Dw  := F_IDLIST_GETREAL( CONCAT(sHead, '_TgtP_Dw'  ), fbIdList );
stConfig.TgtLS_Up := F_IDLIST_GETREAL( CONCAT(sHead, '_TgtLS_Up' ), fbIdList );
stConfig.TgtLS_SUp := F_IDLIST_GETREAL( CONCAT(sHead, '_TgtLS_SUp' ), fbIdList );
stConfig.TgtLS_Dw := F_IDLIST_GETREAL( CONCAT(sHead, '_TgtLS_Dw' ), fbIdList );

stConfig.P_DB     := F_IDLIST_GETREAL( CONCAT(sHead, '_P_DB'     ), fbIdList );
stConfig.LS_DB    := F_IDLIST_GETREAL( CONCAT(sHead, '_LS_DB'    ), fbIdList );
stConfig.LS_Dist  := F_IDLIST_GETREAL( CONCAT(sHead, '_LS_Dist'  ), fbIdList );

stConfig.TimeMax  := F_IDLIST_GETREAL( CONCAT(sHead, '_TimeMax'  ), fbIdList );
stConfig.Delay_Dw := F_IDLIST_GETREAL( CONCAT(sHead, '_Delay_Dw' ), fbIdList );
stConfig.Cycle    := rTime;

stConfig.PP1  := F_IDLIST_GETBOOL( CONCAT(sHead, '_PP1'  ), fbIdList );
stConfig.PP2  := F_IDLIST_GETBOOL( CONCAT(sHead, '_PP2'  ), fbIdList );
stConfig.HP1  := F_IDLIST_GETBOOL( CONCAT(sHead, '_HP1'  ), fbIdList );
stConfig.HP2  := F_IDLIST_GETBOOL( CONCAT(sHead, '_HP2'  ), fbIdList );
stConfig.HP3  := F_IDLIST_GETBOOL( CONCAT(sHead, '_HP3'  ), fbIdList );
END_FUNCTION

(* POU FUN/PARAMETERS/F_READ_MAGIC_DOUBLE_CFG, ST *)
FUNCTION F_READ_MAGIC_DOUBLE_CFG : BOOL
VAR_INPUT
	sHead : STRING;
	rTime : REAL;
END_VAR
VAR_IN_OUT
	stConfig : ST_MAGIC_DOUBLE_CFG;
	fbIdList : FB_IDLIST;
END_VAR
VAR
END_VAR
stConfig.P2Max := F_IDLIST_GETREAL( CONCAT(sHead, '_P2Max' ), fbIdList );
stConfig.P4Max := F_IDLIST_GETREAL( CONCAT(sHead, '_P4Max' ), fbIdList );

stConfig.EVPA4  := F_IDLIST_GETINT( CONCAT(sHead, '_EVPA4' ), fbIdList );
stConfig.EVPA2  := F_IDLIST_GETINT( CONCAT(sHead, '_EVPA2' ), fbIdList );
stConfig.EVPB4  := F_IDLIST_GETINT( CONCAT(sHead, '_EVPB4' ), fbIdList );
stConfig.EVPB2  := F_IDLIST_GETINT( CONCAT(sHead, '_EVPB2' ), fbIdList );
stConfig.EVPFA4 := F_IDLIST_GETINT( CONCAT(sHead, '_EVPFA4' ), fbIdList );
stConfig.EVPFA2 := F_IDLIST_GETINT( CONCAT(sHead, '_EVPFA2' ), fbIdList );
stConfig.EVPFB4 := F_IDLIST_GETINT( CONCAT(sHead, '_EVPFB4' ), fbIdList );
stConfig.EVPFB2 := F_IDLIST_GETINT( CONCAT(sHead, '_EVPFB2' ), fbIdList );

stConfig.EVPRA2 := F_IDLIST_GETINT( CONCAT(sHead, '_EVPRA2' ), fbIdList );
stConfig.EVPRAD := 700;

stConfig.TgtLS4_In  := F_IDLIST_GETREAL( CONCAT(sHead, '_TgtLS4_In'  ), fbIdList );
stConfig.TgtLS4_Out := F_IDLIST_GETREAL( CONCAT(sHead, '_TgtLS4_Out' ), fbIdList );
stConfig.TgtLS2_In  := F_IDLIST_GETREAL( CONCAT(sHead, '_TgtLS2_In'  ), fbIdList );
stConfig.TgtLS2_Out := F_IDLIST_GETREAL( CONCAT(sHead, '_TgtLS2_Out' ), fbIdList );

stConfig.P_DB     := F_IDLIST_GETREAL( CONCAT(sHead, '_P_DB'     ), fbIdList );
stConfig.LS_DB    := F_IDLIST_GETREAL( CONCAT(sHead, '_LS_DB'    ), fbIdList );

stConfig.TimeMax  := F_IDLIST_GETREAL( CONCAT(sHead, '_TimeMax'  ), fbIdList );
stConfig.OutDelay := F_IDLIST_GETREAL( CONCAT(sHead, '_OutDelay' ), fbIdList );
stConfig.EVTDelay := F_IDLIST_GETREAL( CONCAT(sHead, '_EVTDelay' ), fbIdList );
stConfig.Cycle    := rTime;

stConfig.PP1  := F_IDLIST_GETBOOL( CONCAT(sHead, '_PP1'  ), fbIdList );
stConfig.PP2  := F_IDLIST_GETBOOL( CONCAT(sHead, '_PP2'  ), fbIdList );
END_FUNCTION

(* POU FUN/PARAMETERS/F_WRITE_LIFT_KEEL_CFG, ST *)
FUNCTION F_WRITE_LIFT_KEEL_CFG : BOOL
VAR_INPUT
	sHead : STRING;
	wSize   :DWORD;
	pBuffer :POINTER TO BYTE;
END_VAR
VAR_IN_OUT
	wPos     : DWORD;
	stConfig : ST_LIFT_KEEL_CFG;
END_VAR
VAR
END_VAR
F_ADD_STRINGX3_TO_BUFFER( S1:= '$n#', S2:= sHead, S3:=' - Parameters:$n', wSize := wSize, pBuffer := pBuffer, wPos := wPos );

F_ADD_STRINGX4_TO_BUFFER( S1:= CONCAT(sHead, '_PMax_Up' ), S2:='$t', S3:= REAL_TO_STRING( stConfig.PMax_Up ), S4:='$n', wSize := wSize, pBuffer := pBuffer, wPos := wPos );
F_ADD_STRINGX4_TO_BUFFER( S1:= CONCAT(sHead, '_PMax_Dw' ), S2:='$t', S3:= REAL_TO_STRING( stConfig.PMax_Dw ), S4:='$n', wSize := wSize, pBuffer := pBuffer, wPos := wPos );
F_ADD_STRINGX4_TO_BUFFER( S1:= CONCAT(sHead, '_P500_Up' ), S2:='$t', S3:= REAL_TO_STRING( stConfig.P500_Up ), S4:='$n', wSize := wSize, pBuffer := pBuffer, wPos := wPos );
F_ADD_STRINGX4_TO_BUFFER( S1:= CONCAT(sHead, '_P500_Dw' ), S2:='$t', S3:= REAL_TO_STRING( stConfig.P500_Dw ), S4:='$n', wSize := wSize, pBuffer := pBuffer, wPos := wPos );
F_ADD_STRINGX4_TO_BUFFER( S1:= CONCAT(sHead, '_P144_F'  ), S2:='$t', S3:= REAL_TO_STRING( stConfig.P144_F  ), S4:='$n', wSize := wSize, pBuffer := pBuffer, wPos := wPos );
F_ADD_STRINGX4_TO_BUFFER( S1:= CONCAT(sHead, '_P144_S'  ), S2:='$t', S3:= REAL_TO_STRING( stConfig.P144_S  ), S4:='$n', wSize := wSize, pBuffer := pBuffer, wPos := wPos );

F_ADD_STRINGX4_TO_BUFFER( S1:= CONCAT(sHead, '_TgtP_Dw'  ), S2:='$t', S3:= REAL_TO_STRING( stConfig.TgtP_Dw  ), S4:='$n', wSize := wSize, pBuffer := pBuffer, wPos := wPos );
F_ADD_STRINGX4_TO_BUFFER( S1:= CONCAT(sHead, '_TgtLS_Up' ), S2:='$t', S3:= REAL_TO_STRING( stConfig.TgtLS_Up ), S4:='$n', wSize := wSize, pBuffer := pBuffer, wPos := wPos );
F_ADD_STRINGX4_TO_BUFFER( S1:= CONCAT(sHead, '_TgtLS_SUp' ), S2:='$t', S3:= REAL_TO_STRING( stConfig.TgtLS_SUp ), S4:='$n', wSize := wSize, pBuffer := pBuffer, wPos := wPos );
F_ADD_STRINGX4_TO_BUFFER( S1:= CONCAT(sHead, '_TgtLS_Dw' ), S2:='$t', S3:= REAL_TO_STRING( stConfig.TgtLS_Dw ), S4:='$n', wSize := wSize, pBuffer := pBuffer, wPos := wPos );

F_ADD_STRINGX4_TO_BUFFER( S1:= CONCAT(sHead, '_P_DB'     ), S2:='$t', S3:= REAL_TO_STRING( stConfig.P_DB     ), S4:='$n', wSize := wSize, pBuffer := pBuffer, wPos := wPos );
F_ADD_STRINGX4_TO_BUFFER( S1:= CONCAT(sHead, '_LS_DB'    ), S2:='$t', S3:= REAL_TO_STRING( stConfig.LS_DB    ), S4:='$n', wSize := wSize, pBuffer := pBuffer, wPos := wPos );
F_ADD_STRINGX4_TO_BUFFER( S1:= CONCAT(sHead, '_LS_Dist'  ), S2:='$t', S3:= REAL_TO_STRING( stConfig.LS_Dist  ), S4:='$n', wSize := wSize, pBuffer := pBuffer, wPos := wPos );

F_ADD_STRINGX4_TO_BUFFER( S1:= CONCAT(sHead, '_TimeMax'  ), S2:='$t', S3:= REAL_TO_STRING( stConfig.TimeMax  ), S4:='$n', wSize := wSize, pBuffer := pBuffer, wPos := wPos );
F_ADD_STRINGX4_TO_BUFFER( S1:= CONCAT(sHead, '_Delay_Dw' ), S2:='$t', S3:= REAL_TO_STRING( stConfig.Delay_Dw ), S4:='$n', wSize := wSize, pBuffer := pBuffer, wPos := wPos );

F_ADD_STRINGX4_TO_BUFFER( S1:= CONCAT(sHead, '_PP1'  ), S2:='$t', S3:= BOOL_TO_STRING( stConfig.PP1 ), S4:='$n', wSize := wSize, pBuffer := pBuffer, wPos := wPos );
F_ADD_STRINGX4_TO_BUFFER( S1:= CONCAT(sHead, '_PP2'  ), S2:='$t', S3:= BOOL_TO_STRING( stConfig.PP2 ), S4:='$n', wSize := wSize, pBuffer := pBuffer, wPos := wPos );
F_ADD_STRINGX4_TO_BUFFER( S1:= CONCAT(sHead, '_HP1'  ), S2:='$t', S3:= BOOL_TO_STRING( stConfig.HP1 ), S4:='$n', wSize := wSize, pBuffer := pBuffer, wPos := wPos );
F_ADD_STRINGX4_TO_BUFFER( S1:= CONCAT(sHead, '_HP2'  ), S2:='$t', S3:= BOOL_TO_STRING( stConfig.HP2 ), S4:='$n', wSize := wSize, pBuffer := pBuffer, wPos := wPos );
F_ADD_STRINGX4_TO_BUFFER( S1:= CONCAT(sHead, '_HP3'  ), S2:='$t', S3:= BOOL_TO_STRING( stConfig.HP3 ), S4:='$n', wSize := wSize, pBuffer := pBuffer, wPos := wPos );
END_FUNCTION

(* POU FUN/PARAMETERS/F_WRITE_MAGIC_DOUBLE_CFG, ST *)
FUNCTION F_WRITE_MAGIC_DOUBLE_CFG : BOOL
VAR_INPUT
	sHead : STRING;
	wSize   :DWORD;
	pBuffer :POINTER TO BYTE;
END_VAR
VAR_IN_OUT
	wPos     : DWORD;
	stConfig : ST_MAGIC_DOUBLE_CFG;
END_VAR
VAR
END_VAR
F_ADD_STRINGX3_TO_BUFFER( S1:= '$n#', S2:= sHead, S3:=' - Parameters:$n', wSize := wSize, pBuffer := pBuffer, wPos := wPos );

F_ADD_STRINGX4_TO_BUFFER( S1:= CONCAT(sHead, '_P2Max' ), S2:='$t', S3:= REAL_TO_STRING( stConfig.P2Max ), S4:='$n', wSize := wSize, pBuffer := pBuffer, wPos := wPos );
F_ADD_STRINGX4_TO_BUFFER( S1:= CONCAT(sHead, '_P4Max' ), S2:='$t', S3:= REAL_TO_STRING( stConfig.P4Max ), S4:='$n', wSize := wSize, pBuffer := pBuffer, wPos := wPos );

F_ADD_STRINGX4_TO_BUFFER( S1:= CONCAT(sHead, '_EVPA4'   ), S2:='$t', S3:= INT_TO_STRING( stConfig.EVPA4  ), S4:='$n', wSize := wSize, pBuffer := pBuffer, wPos := wPos );
F_ADD_STRINGX4_TO_BUFFER( S1:= CONCAT(sHead, '_EVPA2'   ), S2:='$t', S3:= INT_TO_STRING( stConfig.EVPA2  ), S4:='$n', wSize := wSize, pBuffer := pBuffer, wPos := wPos );
F_ADD_STRINGX4_TO_BUFFER( S1:= CONCAT(sHead, '_EVPB4'   ), S2:='$t', S3:= INT_TO_STRING( stConfig.EVPB4  ), S4:='$n', wSize := wSize, pBuffer := pBuffer, wPos := wPos );
F_ADD_STRINGX4_TO_BUFFER( S1:= CONCAT(sHead, '_EVPB2'   ), S2:='$t', S3:= INT_TO_STRING( stConfig.EVPB2  ), S4:='$n', wSize := wSize, pBuffer := pBuffer, wPos := wPos );
F_ADD_STRINGX4_TO_BUFFER( S1:= CONCAT(sHead, '_EVPFA4'  ), S2:='$t', S3:= INT_TO_STRING( stConfig.EVPFA4 ), S4:='$n', wSize := wSize, pBuffer := pBuffer, wPos := wPos );
F_ADD_STRINGX4_TO_BUFFER( S1:= CONCAT(sHead, '_EVPFA2'  ), S2:='$t', S3:= INT_TO_STRING( stConfig.EVPFA2 ), S4:='$n', wSize := wSize, pBuffer := pBuffer, wPos := wPos );
F_ADD_STRINGX4_TO_BUFFER( S1:= CONCAT(sHead, '_EVPFB4'  ), S2:='$t', S3:= INT_TO_STRING( stConfig.EVPFB4 ), S4:='$n', wSize := wSize, pBuffer := pBuffer, wPos := wPos );
F_ADD_STRINGX4_TO_BUFFER( S1:= CONCAT(sHead, '_EVPFB2'  ), S2:='$t', S3:= INT_TO_STRING( stConfig.EVPFB2 ), S4:='$n', wSize := wSize, pBuffer := pBuffer, wPos := wPos );

F_ADD_STRINGX4_TO_BUFFER( S1:= CONCAT(sHead, '_EVPRA2'  ), S2:='$t', S3:= INT_TO_STRING( stConfig.EVPRA2  ), S4:='$n', wSize := wSize, pBuffer := pBuffer, wPos := wPos );

F_ADD_STRINGX4_TO_BUFFER( S1:= CONCAT(sHead, '_TgtLS4_In'  ), S2:='$t', S3:= REAL_TO_STRING( stConfig.TgtLS4_In  ), S4:='$n', wSize := wSize, pBuffer := pBuffer, wPos := wPos );
F_ADD_STRINGX4_TO_BUFFER( S1:= CONCAT(sHead, '_TgtLS4_Out' ), S2:='$t', S3:= REAL_TO_STRING( stConfig.TgtLS4_Out ), S4:='$n', wSize := wSize, pBuffer := pBuffer, wPos := wPos );
F_ADD_STRINGX4_TO_BUFFER( S1:= CONCAT(sHead, '_TgtLS2_In'  ), S2:='$t', S3:= REAL_TO_STRING( stConfig.TgtLS2_In  ), S4:='$n', wSize := wSize, pBuffer := pBuffer, wPos := wPos );
F_ADD_STRINGX4_TO_BUFFER( S1:= CONCAT(sHead, '_TgtLS2_Out' ), S2:='$t', S3:= REAL_TO_STRING( stConfig.TgtLS2_Out ), S4:='$n', wSize := wSize, pBuffer := pBuffer, wPos := wPos );

F_ADD_STRINGX4_TO_BUFFER( S1:= CONCAT(sHead, '_P_DB'     ), S2:='$t', S3:= REAL_TO_STRING( stConfig.P_DB     ), S4:='$n', wSize := wSize, pBuffer := pBuffer, wPos := wPos );
F_ADD_STRINGX4_TO_BUFFER( S1:= CONCAT(sHead, '_LS_DB'    ), S2:='$t', S3:= REAL_TO_STRING( stConfig.LS_DB    ), S4:='$n', wSize := wSize, pBuffer := pBuffer, wPos := wPos );

F_ADD_STRINGX4_TO_BUFFER( S1:= CONCAT(sHead, '_TimeMax'  ), S2:='$t', S3:= REAL_TO_STRING( stConfig.TimeMax  ), S4:='$n', wSize := wSize, pBuffer := pBuffer, wPos := wPos );
F_ADD_STRINGX4_TO_BUFFER( S1:= CONCAT(sHead, '_OutDelay' ), S2:='$t', S3:= REAL_TO_STRING( stConfig.OutDelay ), S4:='$n', wSize := wSize, pBuffer := pBuffer, wPos := wPos );
F_ADD_STRINGX4_TO_BUFFER( S1:= CONCAT(sHead, '_EVTDelay' ), S2:='$t', S3:= REAL_TO_STRING( stConfig.EVTDelay ), S4:='$n', wSize := wSize, pBuffer := pBuffer, wPos := wPos );

F_ADD_STRINGX4_TO_BUFFER( S1:= CONCAT(sHead, '_PP1'  ), S2:='$t', S3:= BOOL_TO_STRING( stConfig.PP1 ), S4:='$n', wSize := wSize, pBuffer := pBuffer, wPos := wPos );
F_ADD_STRINGX4_TO_BUFFER( S1:= CONCAT(sHead, '_PP2'  ), S2:='$t', S3:= BOOL_TO_STRING( stConfig.PP2 ), S4:='$n', wSize := wSize, pBuffer := pBuffer, wPos := wPos );
END_FUNCTION

(* POU PGN FB/FB_CODE_0000, ST *)
FUNCTION_BLOCK FB_CODE_0000 (*Torque / Speed Control*)
VAR_INPUT
	Enable   : BOOL;
	Source   : BYTE := 16#17;
	Priority : BYTE := 16#06;

	TaskTime     : WORD; (*PLC Taks Time (ms) eg: 10ms*)
	TransmitTime : WORD; (*Synchronous Transmision Time (ms) eg: 100ms*)

	SpeedCtrl  : BOOL;
	TorqueCtrl : BOOL;
	SpeedLimit : REAL;
	TorqueLimit: SINT;
END_VAR
VAR_OUTPUT
	OUT : VARTYPE_EXTCANQUEUE;
	OUT_Enable : BOOL;
END_VAR
VAR
	TimeCnt : WORD;
	dwSrc   : DWORD;
	dwPty   : DWORD;

	bySpeedCtrl  : BYTE;
	byTorqueCtrl : BYTE;
END_VAR
IF Enable THEN
	TimeCnt := TimeCnt + TaskTime;

	IF TransmitTime <= TimeCnt THEN
		TimeCnt := 0;
		dwSrc   := Source;
		dwPty   := Priority AND 16#07;
		dwPty   := SHL( dwPty, 26 );

		bySpeedCtrl  := BOOL_TO_BYTE(SpeedCtrl);
		byTorqueCtrl := BOOL_TO_BYTE(TorqueCtrl) * 2;

		OUT.rxData[0] := bySpeedCtrl OR byTorqueCtrl;

		REAL_TO_BUFFER( pBuffer:= ADR(OUT.rxData[1]), ByteSize := 2, Value:= SpeedLimit, Scale:= 0.125, Offset := 0.0 );

		OUT.rxData[3] := TorqueLimit + 125;
		OUT.rxData[4] := 16#00;
		OUT.rxData[5] := 16#00;
		OUT.rxData[6] := 16#00;
		OUT.rxData[7] := 16#00;

		OUT.length := 8;
		Out.cobId  := 16#80000000 OR dwSrc OR dwPty;
		OUT_Enable := TRUE;
	ELSE
		OUT_Enable := FALSE;

	END_IF
ELSE
	Out_Enable := FALSE;

END_IF
END_FUNCTION_BLOCK

(* POU PGN FB/FB_CODE_F001, ST *)
FUNCTION_BLOCK FB_CODE_F001 (*Electronic Brake Controller*)
VAR_INPUT
	Enable   : BOOL;
	Source   : BYTE := 16#17;
	Priority : BYTE := 16#06;

	TaskTime     : WORD; (*PLC Taks Time (ms) eg: 10ms*)
	TransmitTime : WORD; (*Synchronous Transmision Time (ms) eg: 100ms*)

	EngineStop : BOOL;
END_VAR
VAR_OUTPUT
	OUT : VARTYPE_EXTCANQUEUE;
	OUT_Enable : BOOL;
END_VAR
VAR
	TimeCnt : WORD;
	dwSrc   : DWORD;
	dwPty   : DWORD;
END_VAR
IF Enable THEN
	TimeCnt := TimeCnt + TaskTime;

	IF TransmitTime <= TimeCnt THEN
		TimeCnt := 0;
		dwSrc   := Source;
		dwPty   := Priority AND 16#07;
		dwPty   := SHL( dwPty, 26 );

		OUT.rxData[0] := 16#00;
		OUT.rxData[1] := 16#00;
		OUT.rxData[2] := 16#00;

		IF EngineStop
		THEN OUT.rxData[3] := 16#10;
		ELSE OUT.rxData[3] := 16#00;
		END_IF

		OUT.rxData[4] := 16#00;
		OUT.rxData[5] := 16#00;
		OUT.rxData[6] := 16#00;
		OUT.rxData[7] := 16#00;

		OUT.length := 8;
		Out.cobId  := 16#80F00100 OR dwSrc OR dwPty;
		OUT_Enable := TRUE;
	ELSE
		OUT_Enable := FALSE;

	END_IF
ELSE
	Out_Enable := FALSE;

END_IF
END_FUNCTION_BLOCK

(* POU PGN FB/FB_CODE_F003, ST *)
FUNCTION_BLOCK FB_CODE_F003 (*Torque / Speed Control*)
VAR_INPUT
	Enable   : BOOL;
	Source   : BYTE := 16#31;
	Priority : BYTE := 16#03;

	TaskTime     : WORD; (*PLC Taks Time (ms) eg: 10ms*)
	TransmitTime : WORD; (*Synchronous Transmision Time (ms) eg: 50ms*)

	PedalPerc : REAL;
END_VAR
VAR_OUTPUT
	OUT : VARTYPE_EXTCANQUEUE;
	OUT_Enable : BOOL;
END_VAR
VAR
	TimeCnt : WORD;
	dwSrc   : DWORD;
	dwPty   : DWORD;

	bySpeedCtrl  : BYTE;
	byTorqueCtrl : BYTE;
END_VAR
IF Enable THEN
	TimeCnt := TimeCnt + TaskTime;

	IF TransmitTime <= TimeCnt THEN
		TimeCnt := 0;
		dwSrc   := Source;
		dwPty   := Priority AND 16#07;
		dwPty   := SHL( dwPty, 26 );

		OUT.rxData[0] := 16#00;

		REAL_TO_BUFFER( pBuffer:= ADR(OUT.rxData[1]), ByteSize := 1, Value:= PedalPerc, Scale:= 0.4, Offset := 0.0 );

		OUT.rxData[2] := 16#00;
		OUT.rxData[3] := 16#00;
		OUT.rxData[4] := 16#00;
		OUT.rxData[5] := 16#00;
		OUT.rxData[6] := 16#00;
		OUT.rxData[7] := 16#00;

		OUT.length := 8;
		Out.cobId  := 16#80F00300 OR dwSrc OR dwPty;
		OUT_Enable := TRUE;
	ELSE
		OUT_Enable := FALSE;

	END_IF
ELSE
	Out_Enable := FALSE;

END_IF
END_FUNCTION_BLOCK

(* POU PGN FB/FB_CODE_FF71, ST *)
FUNCTION_BLOCK FB_CODE_FF71 (*Torque / Speed Control*)
VAR_INPUT
	Enable   : BOOL;
	Source   : BYTE := 0;(*16#10;*)
	Priority : BYTE := 16#02;

	TaskTime     : WORD; (*PLC Taks Time (ms) eg: 10ms*)
	TransmitTime : WORD; (*Synchronous Transmision Time (ms) eg: 50ms*)

	PedalPerc  : REAL;
	PedalID    : BYTE;
	PedalFault : BOOL;
END_VAR
VAR_OUTPUT
	OUT : VARTYPE_EXTCANQUEUE;
	OUT_Enable : BOOL;
END_VAR
VAR
	TimeCnt : WORD;
	dwSrc   : DWORD;
	dwPty   : DWORD;

	bySpeedCtrl  : BYTE;
	byTorqueCtrl : BYTE;
END_VAR
IF Enable THEN
	TimeCnt := TimeCnt + TaskTime;

	IF TransmitTime <= TimeCnt THEN
		TimeCnt := 0;
		dwSrc   := Source;
		dwPty   := Priority AND 16#07;
		dwPty   := SHL( dwPty, 26 );

		REAL_TO_BUFFER( pBuffer:= ADR(OUT.rxData[0]), ByteSize := 2, Value:= PedalPerc, Scale:= 0.1, Offset := 0.0 );

		OUT.rxData[2] := PedalID; (*ID*)
		OUT.rxData[3] := 16#00;
		OUT.rxData[3].0 := PedalFault;
		OUT.rxData[4] := 16#00;
		OUT.rxData[5] := 16#00;
		OUT.rxData[6] := 16#00;
		OUT.rxData[7] := 16#00;

		OUT.length := 8;
		Out.cobId  := 16#80FF7100 OR dwSrc OR dwPty;
		OUT_Enable := TRUE;
	ELSE
		OUT_Enable := FALSE;

	END_IF
ELSE
	Out_Enable := FALSE;

END_IF
END_FUNCTION_BLOCK

(* POU PGN FB/FB_DECODE_FEA6, ST *)
FUNCTION_BLOCK FB_DECODE_FEA6
VAR_IN_OUT
	IN: ARRAY [0..7] OF USINT;
END_VAR
VAR_OUTPUT
	FuelTurbocharger1BoostPressure : REAL;
	FuelTurbocharger2BoostPressure : REAL;
	FuelTurbocharger3BoostPressure : REAL;
	FuelTurbocharger4BoostPressure : REAL;

	Count : DWORD;
END_VAR
VAR
	Debug : BOOL;
	Buffer: ARRAY [0..7] OF USINT;
END_VAR
FuelTurbocharger1BoostPressure := BUFFER_TO_REAL( pBuffer:= ADR(IN[0]), ByteSize := 2, Scale:= 0.125, Offset := 0.0 );
FuelTurbocharger2BoostPressure := BUFFER_TO_REAL( pBuffer:= ADR(IN[2]), ByteSize := 2, Scale:= 0.125, Offset := 0.0 );
FuelTurbocharger3BoostPressure := BUFFER_TO_REAL( pBuffer:= ADR(IN[4]), ByteSize := 2, Scale:= 0.125, Offset := 0.0 );
FuelTurbocharger4BoostPressure := BUFFER_TO_REAL( pBuffer:= ADR(IN[6]), ByteSize := 2, Scale:= 0.125, Offset := 0.0 );

Count := Count + 1;

IF Debug THEN MEMCPY(destAddr := ADR(Buffer), srcAddr := ADR(IN), n := 8); END_IF
END_FUNCTION_BLOCK

(* POU PGN FB/FB_DECODE_FECA, ST *)
FUNCTION_BLOCK FB_DECODE_FECA (*DM1 (diagnostic message 1)*)
VAR_IN_OUT
	IN: ARRAY [0..7] OF USINT;
END_VAR
VAR_OUTPUT
	EngineInjectorMeteringRail1Pressure : REAL;

	Count : DWORD;
END_VAR
VAR
	Debug : BOOL;
	Buffer: ARRAY [0..7] OF USINT;
END_VAR
EngineInjectorMeteringRail1Pressure  := BUFFER_TO_REAL( pBuffer:= ADR(IN[2]), ByteSize := 2, Scale:= 0.00390625, Offset:= 0.0 );

Count := Count + 1;

IF Debug THEN MEMCPY(destAddr := ADR(Buffer), srcAddr := ADR(IN), n := 8); END_IF
END_FUNCTION_BLOCK

(* POU PGN FB/FB_DECODE_FEF6_VM, ST *)
FUNCTION_BLOCK FB_DECODE_FEF6_VM
VAR_IN_OUT
	IN: ARRAY [0..7] OF USINT;
END_VAR
VAR_OUTPUT
	EngineBoostPressure : REAL;

	Count : DWORD;
END_VAR
EngineBoostPressure := BUFFER_TO_REAL( pBuffer:= ADR(IN[1]), ByteSize := 1, Scale:= 2.0, Offset := 0.0 );

Count := Count + 1;
END_FUNCTION_BLOCK

(* Visualisation VISU_0_MAIN
ellipse at (195,415)-(216,436): text "P"; alarm colour if MAIN.fbBoard.LS_P_Out
rectangle at (20,0)-(461,51): text "HOME %s"; shows MAIN.LoadLabel
rectangle at (20,550)-(526,601): text "%s"; shows INPUTS.sVisuTime
ellipse at (375,70)-(436,131): text "SHUT / DOWN"; alarm colour if MAIN.HMI_ShutDw; taps MAIN.HMI_ShutDw
ellipse at (460,70)-(521,131): text "ENABLE"; shows MAIN.SysPass; alarm colour if MAIN.HMI_Enable; taps MAIN.HMI_Enable
rectangle at (600,255)-(851,276): text "Propulsion: 		%.0f RPM"; shows .Prop_RPM; runs INTERN ASSIGN INPUTS.PresSelCalStbd[9]:=(FALSE)
rectangle at (335,135)-(561,206): text "%s"; shows MAIN.SysLabel; dynamic style MAIN.SysColor
rectangle at (0,0)-(1,1): text "{ExtendedElement},Visu\ElementDLL.ete,0,@Zeigerinstrument,221,220,-40,1,0,0,128,1,RECV_J1939.F004.EngineActualSpeed,RPM,%.0f,0,0,0,200,600,0,3000,0,0,0,0,0,0,0,-13,100,700,MS Sans Serif,1,5,0,600,255,0,0,800,2400,0,255,0,2400,2800,255,255,0,2800,3000,255,0,0,600,800,255,255,0,0,255,255,255,,"
rectangle at (35,162)-(43,178): text "0"
rectangle at (8,83)-(32,99): text "600"
rectangle at (54,19)-(86,35): text "1200"
rectangle at (135,19)-(167,35): text "1800"
rectangle at (185,83)-(217,99): text "2400"
rectangle at (166,162)-(198,178): text "3000"
rectangle at (94,116)-(127,132): text "RPM"
polygon at (107,61)-(115,111): angle ((RECV_J1939.F004.EngineActualSpeed * 1.0)-1500) * 0.0866667
polygon at (109,49)-(112,57): angle ((RECV_J1939.F004.EngineActualSpeed * 1.0)-1500) * 0.0866667
rectangle at (650,190)-(716,211): text "%.0f"; shows RECV_J1939.F004.EngineActualSpeed
rounded rectangle at (900,490)-(1021,551): alarm colour if ALARMS.Adver
rounded rectangle at (905,495)-(1016,546): text "ALARMS"; opens VISU_1_ALARMS
rounded rectangle at (900,160)-(1021,211): alarm colour if ALARMS.EngAdver
rounded rectangle at (905,165)-(1016,206): text "ENGINE && / PROPULSION"; opens VISU_1_ENGINE
rounded rectangle at (900,105)-(1021,156): alarm colour if ALARMS.PumpAdver
rounded rectangle at (905,110)-(1016,151): text "PUMPS"; opens VISU_1_PUMPS
rounded rectangle at (900,50)-(1021,101): alarm colour if ALARMS.TankAdver
rounded rectangle at (905,55)-(1016,96): text "TANK"; opens VISU_1_TANK
rounded rectangle at (905,220)-(1016,261): text "WINCHES"; opens VISU_1_WINCHES
rounded rectangle at (905,275)-(1016,316): text "CYLINDERS"; opens VISU_1_CYLINDERS1
rounded rectangle at (905,330)-(1016,371): text "SPECIAL / FUNCTIONS"; opens VISU_1_SPECIAL
rounded rectangle at (905,385)-(1016,426): text "KEEL && / BOARD"; opens VISU_1_KEEL
rounded rectangle at (905,440)-(1016,481): text "WATER / BALLAST"; opens VISU_1_WB
rounded rectangle at (345,395)-(416,466): alarm colour if OUTPUTS.byDimmerState > 0
ellipse at (350,400)-(411,461): text "DIMMER"; alarm colour if OUTPUTS.SIDimmerUp.In; taps OUTPUTS.SIDimmerUp.In
rectangle at (420,395)-(481,416): text "PANELS"
rectangle at (485,420)-(551,441): text "%d %%"; shows OUTPUTS.Dimmer_Ledbar; editable 1..100
rectangle at (420,420)-(481,441): text "LEDBARS"
rectangle at (485,395)-(551,416): text "%d %%"; shows OUTPUTS.Dimmer_Panels; editable 0..100
rectangle at (420,445)-(481,466): text "WINCHES"
rectangle at (485,445)-(551,466): text "%d %%"; shows OUTPUTS.Dimmer_Decklink; editable 1..100
rectangle at (10,485)-(446,501): text "%s"; shows ALARMS.AlarmList[1]; alarm colour if ALARMS.AlarmFlag[1]
rectangle at (10,500)-(446,516): text "%s"; shows ALARMS.AlarmList[2]; alarm colour if ALARMS.AlarmFlag[2]
rectangle at (10,515)-(446,531): text "%s"; shows ALARMS.AlarmList[3]; alarm colour if ALARMS.AlarmFlag[3]
rectangle at (10,530)-(446,546): text "%s"; shows ALARMS.AlarmList[4]; alarm colour if ALARMS.AlarmFlag[4]
rectangle at (455,485)-(891,501): text "%s"; shows ALARMS.AlarmList[5]; alarm colour if ALARMS.AlarmFlag[5]
rectangle at (455,500)-(891,516): text "%s"; shows ALARMS.AlarmList[6]; alarm colour if ALARMS.AlarmFlag[6]
rectangle at (455,515)-(891,531): text "%s"; shows ALARMS.AlarmList[7]; alarm colour if ALARMS.AlarmFlag[7]
rectangle at (455,530)-(891,546): text "%s"; shows ALARMS.AlarmList[8]; alarm colour if ALARMS.AlarmFlag[8]
rectangle at (0,0)-(1,1): text "{ExtendedElement},Visu\ElementDLL.ete,1,@Bargraph,91,151,1,1,0,RECV_J1939.F004.EngineActualTorque,, %.0f,12.5,25,0,100,0,0,0,0,0,0,0,-13,100,700,MS Sans Serif,0,255,0,255,0,0,0,0,0,0,0,0,0,,1,"
rectangle at (15,75)-(34,140): alarm colour if (RECV_J1939.F004.EngineActualTorque) < 0; top ((RECV_J1939.F004.EngineActualTorque * 1.0) - 50)  * -1.3
rectangle at (35,129)-(84,150): text "0"
rectangle at (35,97)-(84,118): text "25"
rectangle at (35,64)-(84,85): text "50"
rectangle at (35,32)-(84,53): text "75"
rectangle at (35,0)-(84,20): text "100"
rectangle at (800,220)-(871,241): text "%d %%"; shows RECV_J1939.F004.EngineActualTorque
ellipse at (650,215)-(716,236): text "PROP."; alarm colour if ENGINE.Propulion_ON
rectangle at (600,280)-(851,301): text "Coolant Temperature:	%.0f ºC"; shows RECV_J1939.FEEE.EngineCoolantTemperature
rectangle at (600,300)-(851,321): text "Fuel Temperature:	%.0f ºC"; shows RECV_J1939.FEEE.EngineFuelTemperature
rectangle at (600,325)-(851,346): text "Fuel Pressure:		%.0f MPa"; shows RECV_J1939.FEDB.EngineInjectorMeteringRail1Pressure
rectangle at (600,345)-(851,366): text "Engine Oil Pressure:	%.0f kPa"; shows RECV_J1939.FEEF.EngineOilPressure
rectangle at (600,365)-(851,386): text "Air Intake Pressure:	%.0f kPa"; shows RECV_J1939.FEF6.EngineIntakeMF1Pressure
rectangle at (600,390)-(851,411): text "Electrical Potential:	%.1f V"; shows RECV_J1939.FEF7.ElectricalPotential
rectangle at (600,415)-(851,436): text "Engine Fuel Rate:	%.1f L/h"; shows RECV_J1939.FEF2.EngineFuelRate
rectangle at (600,435)-(851,456): text "Total Hours:		%.1f hr"; shows RECV_J1939.FEE5.EngineTotalHoursOfOperation
rectangle at (45,75)-(296,96): text "Hydro Oil Temperature:	%.0f ºC"; shows .S011.Deg; alarm colour if .S011.Alarm.Alarm
rectangle at (685,50)-(766,71): text "ENGINE"
rectangle at (130,50)-(211,71): text "HYDRO"
rectangle at (45,125)-(296,146): text "LP Line P101:		%.0f bar"; shows P101.Bar; alarm colour if P101.Alarm.Alarm
rectangle at (45,145)-(296,166): text "LP Line P201:		%.0f bar"; shows P201.Bar; alarm colour if P201.Alarm.Alarm
rectangle at (45,165)-(296,186): text "HP Line P103:		%.0f bar"; shows P103.Bar; alarm colour if P103.Alarm.Alarm
rectangle at (45,190)-(296,211): text "GS A Line P001:	%.0f bar"; shows P001.Bar; alarm colour if P001.Alarm.Alarm
rectangle at (45,210)-(296,231): text "GS B Line P002:		%.0f bar"; shows P002.Bar; alarm colour if P002.Alarm.Alarm
rectangle at (45,315)-(296,336): text "HP Functions in use:	%d"; shows POWERPACK.NHP
rectangle at (45,295)-(296,316): text "LP Functions in use:	%d"; shows POWERPACK.NLP
rectangle at (45,275)-(296,296): text "Winches in use:		%d"; shows POWERPACK.NW
rectangle at (115,250)-(226,271): text "FUNCTIONS"
ellipse at (275,345)-(296,366): text "S"; alarm colour if MAIN.fbKeel.KEEL_I
ellipse at (195,345)-(216,366): text "P"; alarm colour if MAIN.fbKeel.KEEL_O
ellipse at (235,345)-(256,366): text "C"; alarm colour if MAIN.fbKeel.KEEL_C
ellipse at (215,350)-(236,366): text "SP"; alarm colour if MAIN.fbKeel.KEEL_SO
ellipse at (255,350)-(276,366): text "SS"; alarm colour if MAIN.fbKeel.KEEL_SI
rectangle at (45,345)-(176,366): text "Keel:	%.1f %%"; shows MAIN.fbKeel.LS_Pos; alarm colour if MAIN.fbKeel.LS_Err
rectangle at (45,415)-(176,436): text "Dgb P.:	%.1f %%"; shows LS801.Pos; alarm colour if LS801.Alarm.Alarm
rectangle at (45,435)-(176,456): text "Dgb S.:	%.1f %%"; shows LS803.Pos; alarm colour if LS803.Alarm.Alarm
ellipse at (235,415)-(256,436): text "C"; alarm colour if MAIN.fbBoard.LS_P_Mid
ellipse at (195,435)-(216,456): text "P"; alarm colour if MAIN.fbBoard.LS_S_In
ellipse at (275,435)-(296,456): text "S"; alarm colour if MAIN.fbBoard.LS_S_Out
ellipse at (235,435)-(256,456): text "C"; alarm colour if MAIN.fbBoard.LS_S_Mid
ellipse at (275,415)-(296,436): text "S"; alarm colour if MAIN.fbBoard.LS_P_In
ellipse at (255,440)-(276,456): text "SS"; alarm colour if MAIN.fbBoard.LS_Safe_S_Out
ellipse at (215,440)-(236,456): text "SP"; alarm colour if MAIN.fbBoard.LS_Safe_S_In
ellipse at (255,420)-(276,436): text "SS"; alarm colour if MAIN.fbBoard.LS_Safe_P_In
ellipse at (215,420)-(236,436): text "SP"; alarm colour if MAIN.fbBoard.LS_Safe_P_Out
rectangle at (45,365)-(296,386): text "Keel P. P1001:		%.0f bar"; shows P1001.Bar; alarm colour if P1001.Alarm.Alarm
rectangle at (45,385)-(296,406): text "Keel S. P1002:		%.0f bar"; shows P1002.Bar; alarm colour if P1002.Alarm.Alarm
rectangle at (45,100)-(296,121): text "Oil Tank P010:		%.0f bar"; shows P010.Bar; alarm colour if P010.Alarm.Alarm
42 more shapes without text or variables
*)

(* Visualisation VISU_1_ALARMS
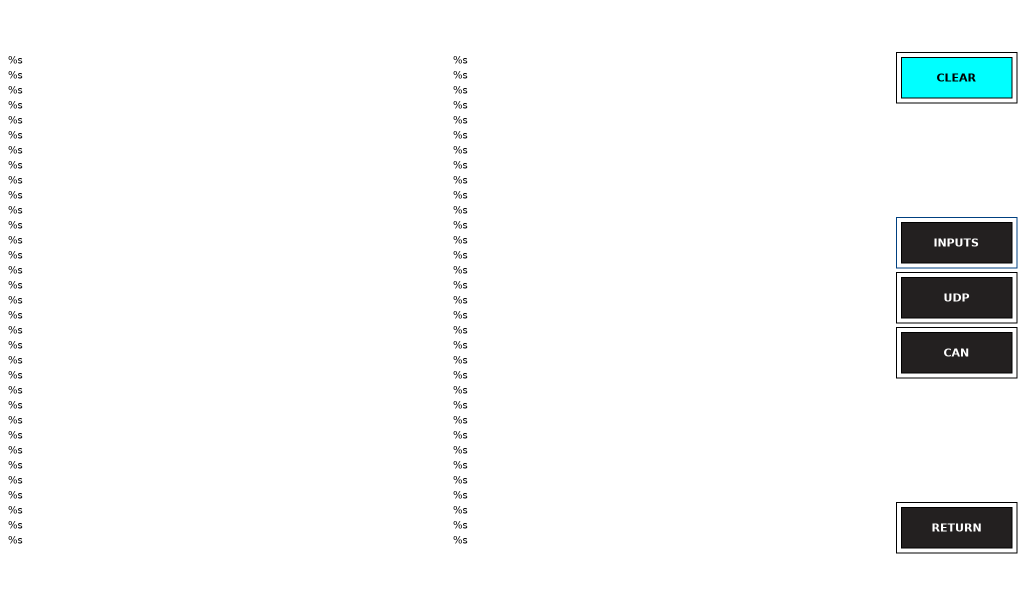
rounded rectangle at (900,325)-(1021,376): alarm colour if ALARMS.CanAdver
rectangle at (20,0)-(331,51): text "ALARMS"
rectangle at (15,550)-(326,601): text "%s"; shows INPUTS.sVisuTime
rectangle at (10,50)-(446,66): text "%s"; shows ALARMS.AlarmList[1]; alarm colour if ALARMS.AlarmFlag[1]
rectangle at (10,65)-(446,81): text "%s"; shows ALARMS.AlarmList[2]; alarm colour if ALARMS.AlarmFlag[2]
rectangle at (10,80)-(446,96): text "%s"; shows ALARMS.AlarmList[3]; alarm colour if ALARMS.AlarmFlag[3]
rectangle at (10,95)-(446,111): text "%s"; shows ALARMS.AlarmList[4]; alarm colour if ALARMS.AlarmFlag[4]
rectangle at (10,110)-(446,126): text "%s"; shows ALARMS.AlarmList[5]; alarm colour if ALARMS.AlarmFlag[5]
rectangle at (10,125)-(446,141): text "%s"; shows ALARMS.AlarmList[6]; alarm colour if ALARMS.AlarmFlag[6]
rectangle at (10,140)-(446,156): text "%s"; shows ALARMS.AlarmList[7]; alarm colour if ALARMS.AlarmFlag[7]
rectangle at (10,155)-(446,171): text "%s"; shows ALARMS.AlarmList[8]; alarm colour if ALARMS.AlarmFlag[8]
rectangle at (10,170)-(446,186): text "%s"; shows ALARMS.AlarmList[9]; alarm colour if ALARMS.AlarmFlag[9]
rectangle at (10,185)-(446,201): text "%s"; shows ALARMS.AlarmList[10]; alarm colour if ALARMS.AlarmFlag[10]
rounded rectangle at (905,505)-(1016,546): text "RETURN"; opens VISU_0_MAIN
rounded rectangle at (905,330)-(1016,371): text "CAN"; opens VISU_2_CAN
rounded rectangle at (900,270)-(1021,321): alarm colour if TOFARO.fbUdpSend.bError
rounded rectangle at (905,275)-(1016,316): text "UDP"; opens VISU_2_UDP
rounded rectangle at (905,220)-(1016,261): text "INPUTS"; opens VISU_2_INPUTS
rectangle at (10,200)-(446,216): text "%s"; shows ALARMS.AlarmList[11]; alarm colour if ALARMS.AlarmFlag[11]
rectangle at (10,215)-(446,231): text "%s"; shows ALARMS.AlarmList[12]; alarm colour if ALARMS.AlarmFlag[12]
rectangle at (10,230)-(446,246): text "%s"; shows ALARMS.AlarmList[13]; alarm colour if ALARMS.AlarmFlag[13]
rectangle at (10,245)-(446,261): text "%s"; shows ALARMS.AlarmList[14]; alarm colour if ALARMS.AlarmFlag[14]
rectangle at (10,260)-(446,276): text "%s"; shows ALARMS.AlarmList[15]; alarm colour if ALARMS.AlarmFlag[15]
rectangle at (10,275)-(446,291): text "%s"; shows ALARMS.AlarmList[16]; alarm colour if ALARMS.AlarmFlag[16]
rectangle at (10,290)-(446,306): text "%s"; shows ALARMS.AlarmList[17]; alarm colour if ALARMS.AlarmFlag[17]
rectangle at (10,305)-(446,321): text "%s"; shows ALARMS.AlarmList[18]; alarm colour if ALARMS.AlarmFlag[18]
rectangle at (10,320)-(446,336): text "%s"; shows ALARMS.AlarmList[19]; alarm colour if ALARMS.AlarmFlag[19]
rectangle at (10,335)-(446,351): text "%s"; shows ALARMS.AlarmList[20]; alarm colour if ALARMS.AlarmFlag[20]
rectangle at (10,350)-(446,366): text "%s"; shows ALARMS.AlarmList[21]; alarm colour if ALARMS.AlarmFlag[21]
rectangle at (10,365)-(446,381): text "%s"; shows ALARMS.AlarmList[22]; alarm colour if ALARMS.AlarmFlag[22]
rectangle at (10,380)-(446,396): text "%s"; shows ALARMS.AlarmList[23]; alarm colour if ALARMS.AlarmFlag[23]
rectangle at (10,395)-(446,411): text "%s"; shows ALARMS.AlarmList[24]; alarm colour if ALARMS.AlarmFlag[24]
rectangle at (10,410)-(446,426): text "%s"; shows ALARMS.AlarmList[25]; alarm colour if ALARMS.AlarmFlag[25]
rectangle at (10,425)-(446,441): text "%s"; shows ALARMS.AlarmList[26]; alarm colour if ALARMS.AlarmFlag[26]
rectangle at (10,440)-(446,456): text "%s"; shows ALARMS.AlarmList[27]; alarm colour if ALARMS.AlarmFlag[27]
rectangle at (10,455)-(446,471): text "%s"; shows ALARMS.AlarmList[28]; alarm colour if ALARMS.AlarmFlag[28]
rectangle at (10,470)-(446,486): text "%s"; shows ALARMS.AlarmList[29]; alarm colour if ALARMS.AlarmFlag[29]
rectangle at (10,485)-(446,501): text "%s"; shows ALARMS.AlarmList[30]; alarm colour if ALARMS.AlarmFlag[30]
rectangle at (10,500)-(446,516): text "%s"; shows ALARMS.AlarmList[31]; alarm colour if ALARMS.AlarmFlag[31]
rectangle at (10,515)-(446,531): text "%s"; shows ALARMS.AlarmList[32]; alarm colour if ALARMS.AlarmFlag[32]
rectangle at (10,530)-(446,546): text "%s"; shows ALARMS.AlarmList[33]; alarm colour if ALARMS.AlarmFlag[33]
rectangle at (455,50)-(891,66): text "%s"; shows ALARMS.AlarmList[34]; alarm colour if ALARMS.AlarmFlag[34]
rectangle at (455,65)-(891,81): text "%s"; shows ALARMS.AlarmList[35]; alarm colour if ALARMS.AlarmFlag[35]
rectangle at (455,80)-(891,96): text "%s"; shows ALARMS.AlarmList[36]; alarm colour if ALARMS.AlarmFlag[36]
rectangle at (455,95)-(891,111): text "%s"; shows ALARMS.AlarmList[37]; alarm colour if ALARMS.AlarmFlag[37]
rectangle at (455,110)-(891,126): text "%s"; shows ALARMS.AlarmList[38]; alarm colour if ALARMS.AlarmFlag[38]
rectangle at (455,125)-(891,141): text "%s"; shows ALARMS.AlarmList[39]; alarm colour if ALARMS.AlarmFlag[39]
rectangle at (455,140)-(891,156): text "%s"; shows ALARMS.AlarmList[40]; alarm colour if ALARMS.AlarmFlag[40]
rectangle at (455,155)-(891,171): text "%s"; shows ALARMS.AlarmList[41]; alarm colour if ALARMS.AlarmFlag[41]
rectangle at (455,170)-(891,186): text "%s"; shows ALARMS.AlarmList[42]; alarm colour if ALARMS.AlarmFlag[42]
rectangle at (455,185)-(891,201): text "%s"; shows ALARMS.AlarmList[43]; alarm colour if ALARMS.AlarmFlag[43]
rectangle at (455,200)-(891,216): text "%s"; shows ALARMS.AlarmList[44]; alarm colour if ALARMS.AlarmFlag[44]
rectangle at (455,215)-(891,231): text "%s"; shows ALARMS.AlarmList[45]; alarm colour if ALARMS.AlarmFlag[45]
rectangle at (455,230)-(891,246): text "%s"; shows ALARMS.AlarmList[46]; alarm colour if ALARMS.AlarmFlag[46]
rectangle at (455,245)-(891,261): text "%s"; shows ALARMS.AlarmList[47]; alarm colour if ALARMS.AlarmFlag[47]
rectangle at (455,260)-(891,276): text "%s"; shows ALARMS.AlarmList[48]; alarm colour if ALARMS.AlarmFlag[48]
rectangle at (455,275)-(891,291): text "%s"; shows ALARMS.AlarmList[49]; alarm colour if ALARMS.AlarmFlag[49]
rectangle at (455,290)-(891,306): text "%s"; shows ALARMS.AlarmList[50]; alarm colour if ALARMS.AlarmFlag[50]
rectangle at (455,305)-(891,321): text "%s"; shows ALARMS.AlarmList[51]; alarm colour if ALARMS.AlarmFlag[51]
rectangle at (455,320)-(891,336): text "%s"; shows ALARMS.AlarmList[52]; alarm colour if ALARMS.AlarmFlag[52]
rectangle at (455,335)-(891,351): text "%s"; shows ALARMS.AlarmList[53]; alarm colour if ALARMS.AlarmFlag[53]
rectangle at (455,350)-(891,366): text "%s"; shows ALARMS.AlarmList[54]; alarm colour if ALARMS.AlarmFlag[54]
rectangle at (455,365)-(891,381): text "%s"; shows ALARMS.AlarmList[55]; alarm colour if ALARMS.AlarmFlag[55]
rectangle at (455,380)-(891,396): text "%s"; shows ALARMS.AlarmList[56]; alarm colour if ALARMS.AlarmFlag[56]
rectangle at (455,395)-(891,411): text "%s"; shows ALARMS.AlarmList[57]; alarm colour if ALARMS.AlarmFlag[57]
rectangle at (455,410)-(891,426): text "%s"; shows ALARMS.AlarmList[58]; alarm colour if ALARMS.AlarmFlag[58]
rectangle at (455,425)-(891,441): text "%s"; shows ALARMS.AlarmList[59]; alarm colour if ALARMS.AlarmFlag[59]
rectangle at (455,440)-(891,456): text "%s"; shows ALARMS.AlarmList[60]; alarm colour if ALARMS.AlarmFlag[60]
rectangle at (455,455)-(891,471): text "%s"; shows ALARMS.AlarmList[61]; alarm colour if ALARMS.AlarmFlag[61]
rectangle at (455,470)-(891,486): text "%s"; shows ALARMS.AlarmList[62]; alarm colour if ALARMS.AlarmFlag[62]
rectangle at (455,485)-(891,501): text "%s"; shows ALARMS.AlarmList[63]; alarm colour if ALARMS.AlarmFlag[63]
rectangle at (455,500)-(891,516): text "%s"; shows ALARMS.AlarmList[64]; alarm colour if ALARMS.AlarmFlag[64]
rectangle at (455,515)-(891,531): text "%s"; shows ALARMS.AlarmList[65]; alarm colour if ALARMS.AlarmFlag[65]
rectangle at (455,530)-(891,546): text "%s"; shows ALARMS.AlarmList[66]; alarm colour if ALARMS.AlarmFlag[66]
rounded rectangle at (905,55)-(1016,96): text "CLEAR"; alarm colour if ALARMS.Clear; taps ALARMS.Clear
3 more shapes without text or variables
*)

(* Visualisation VISU_1_CYLINDERS1
rectangle at (20,550)-(331,601): text "%s"; shows INPUTS.sVisuTime
rounded rectangle at (905,505)-(1016,546): text "RETURN"; opens VISU_0_MAIN
rectangle at (20,0)-(331,51): text "CYLINDERS 1"
rectangle at (35,350)-(116,371): text "%.0f bar"; shows P301.Bar; alarm colour if P301.Alarm.Adver; runs INTERN ASSIGN INPUTS.PresSelCalStbd[9]:=(FALSE)
rectangle at (35,430)-(116,451): text "%.1f %%"; shows LS301.Pos; alarm colour if LS301.Alarm.Adver; runs INTERN ASSIGN INPUTS.PresSelCalStbd[9]:=(FALSE)
rectangle at (35,390)-(116,411): text "%.0f Kg"; shows L301.Kg; runs INTERN ASSIGN INPUTS.PresSelCalStbd[9]:=(FALSE)
rectangle at (0,0)-(1,1): text "{ExtendedElement},Visu\ElementDLL.ete,1,@Bargraph,86,21,3,0,0,LS301.Pos,,%,25,50,0,100,0,0,0,0,0,0,0,-13,16,700,Arial,0,255,0,255,0,0,0,0,0,0,0,0,0,,0,"
rectangle at (0,0)-(44,21): alarm colour if (LS301.Pos) < 0; right ((LS301.Pos * 1.0) - 50)  * 0.86
ellipse at (40,165)-(111,236): alarm colour if MAIN.fbSE301.OUT_CylIn
ellipse at (40,245)-(111,316): alarm colour if MAIN.fbSE301.OUT_CylOut
ellipse at (50,175)-(101,226): text "IN"; alarm colour if MAIN.fbSE301.IN_Hmi_CylIn; taps MAIN.fbSE301.IN_Hmi_CylIn
ellipse at (50,255)-(101,306): text "OUT"; alarm colour if MAIN.fbSE301.IN_Hmi_CylOut; taps MAIN.fbSE301.IN_Hmi_CylOut
rectangle at (35,335)-(106,351): text "P301"
rectangle at (35,375)-(106,391): text "L301"
rectangle at (35,415)-(106,431): text "LS301"
ellipse at (35,485)-(76,506): text "IN"; alarm colour if MAIN.fbSE301.LS_In
ellipse at (75,485)-(116,506): text "OUT"; alarm colour if MAIN.fbSE301.LS_Out
rectangle at (685,350)-(766,371): text "%.0f bar"; shows P901.Bar; alarm colour if P901.Alarm.Adver; runs INTERN ASSIGN INPUTS.PresSelCalStbd[9]:=(FALSE)
rectangle at (685,430)-(766,451): text "%.1f %%"; shows LS901.Pos; alarm colour if LS901.Alarm.Adver; runs INTERN ASSIGN INPUTS.PresSelCalStbd[9]:=(FALSE)
rectangle at (685,390)-(766,411): text "%.0f Kg"; shows L901.Kg; runs INTERN ASSIGN INPUTS.PresSelCalStbd[9]:=(FALSE)
rectangle at (0,0)-(1,1): text "{ExtendedElement},Visu\ElementDLL.ete,1,@Bargraph,86,21,3,0,0,LS901.Pos,,%,25,50,0,100,0,0,0,0,0,0,0,-13,16,700,Arial,0,255,0,255,0,0,0,0,0,0,0,0,0,,0,"
rectangle at (0,0)-(44,21): alarm colour if (LS901.Pos) < 0; right ((LS901.Pos * 1.0) - 50)  * 0.86
ellipse at (690,165)-(761,236): alarm colour if MAIN.fbBSY.OUT_P_In
ellipse at (690,245)-(761,316): alarm colour if MAIN.fbBSY.OUT_P_Out
ellipse at (700,175)-(751,226): text "IN"; alarm colour if MAIN.fbBSY.IN_Hmi_P_In; taps MAIN.fbBSY.IN_Hmi_P_In
ellipse at (700,255)-(751,306): text "OUT"; alarm colour if MAIN.fbBSY.IN_Hmi_P_Out; taps MAIN.fbBSY.IN_Hmi_P_Out
rectangle at (685,335)-(756,351): text "P901"
rectangle at (685,375)-(756,391): text "L901"
rectangle at (685,415)-(756,431): text "LS901"
ellipse at (685,485)-(726,506): text "IN"; alarm colour if MAIN.fbBSY.LS_P_In
ellipse at (725,485)-(766,506): text "OUT"; alarm colour if MAIN.fbBSY.LS_P_Out
rectangle at (135,350)-(216,371): text "%.0f bar"; shows P303.Bar; alarm colour if P303.Alarm.Adver; runs INTERN ASSIGN INPUTS.PresSelCalStbd[9]:=(FALSE)
rectangle at (135,430)-(216,451): text "%.1f %%"; shows LS303.Pos; alarm colour if LS303.Alarm.Adver; runs INTERN ASSIGN INPUTS.PresSelCalStbd[9]:=(FALSE)
rectangle at (135,390)-(216,411): text "%.0f Kg"; shows L303.Kg; runs INTERN ASSIGN INPUTS.PresSelCalStbd[9]:=(FALSE)
rectangle at (0,0)-(1,1): text "{ExtendedElement},Visu\ElementDLL.ete,1,@Bargraph,86,21,3,0,0,LS303.Pos,,%,25,50,0,100,0,0,0,0,0,0,0,-13,16,700,Arial,0,255,0,255,0,0,0,0,0,0,0,0,0,,0,"
rectangle at (0,0)-(44,21): alarm colour if (LS303.Pos) < 0; right ((LS303.Pos * 1.0) - 50)  * 0.86
ellipse at (140,165)-(211,236): alarm colour if MAIN.fbSE303.OUT_CylIn
ellipse at (140,245)-(211,316): alarm colour if MAIN.fbSE303.OUT_CylOut
ellipse at (150,175)-(201,226): text "IN"; alarm colour if MAIN.fbSE303.IN_Hmi_CylIn; taps MAIN.fbSE303.IN_Hmi_CylIn
ellipse at (150,255)-(201,306): text "OUT"; alarm colour if MAIN.fbSE303.IN_Hmi_CylOut; taps MAIN.fbSE303.IN_Hmi_CylOut
rectangle at (135,335)-(206,351): text "P303"
rectangle at (135,375)-(206,391): text "L303"
rectangle at (135,415)-(206,431): text "LS303"
ellipse at (135,485)-(176,506): text "IN"; alarm colour if MAIN.fbSE303.LS_In
ellipse at (175,485)-(216,506): text "OUT"; alarm colour if MAIN.fbSE303.LS_Out
rectangle at (245,350)-(326,371): text "%.0f bar"; shows P305.Bar; alarm colour if P305.Alarm.Adver; runs INTERN ASSIGN INPUTS.PresSelCalStbd[9]:=(FALSE)
rectangle at (245,430)-(326,451): text "%.1f %%"; shows LS305.Pos; alarm colour if LS305.Alarm.Adver; runs INTERN ASSIGN INPUTS.PresSelCalStbd[9]:=(FALSE)
rectangle at (245,390)-(326,411): text "%.0f Kg"; shows L305.Kg; runs INTERN ASSIGN INPUTS.PresSelCalStbd[9]:=(FALSE)
rectangle at (0,0)-(1,1): text "{ExtendedElement},Visu\ElementDLL.ete,1,@Bargraph,86,21,3,0,0,LS305.Pos,,%,25,50,0,100,0,0,0,0,0,0,0,-13,16,700,Arial,0,255,0,255,0,0,0,0,0,0,0,0,0,,0,"
rectangle at (0,0)-(44,21): alarm colour if (LS305.Pos) < 0; right ((LS305.Pos * 1.0) - 50)  * 0.86
ellipse at (250,165)-(321,236): alarm colour if MAIN.fbSE305.OUT_CylIn
ellipse at (250,245)-(321,316): alarm colour if MAIN.fbSE305.OUT_CylOut
ellipse at (260,175)-(311,226): text "IN"; alarm colour if MAIN.fbSE305.IN_Hmi_CylIn; taps MAIN.fbSE305.IN_Hmi_CylIn
ellipse at (260,255)-(311,306): text "OUT"; alarm colour if MAIN.fbSE305.IN_Hmi_CylOut; taps MAIN.fbSE305.IN_Hmi_CylOut
rectangle at (260,60)-(311,81): text "J5"
rectangle at (245,335)-(316,351): text "P305"
rectangle at (245,375)-(316,391): text "L305"
rectangle at (245,415)-(316,431): text "LS305"
ellipse at (245,485)-(286,506): text "IN"; alarm colour if MAIN.fbSE305.LS_In
ellipse at (285,485)-(326,506): text "OUT"; alarm colour if MAIN.fbSE305.LS_Out
rectangle at (355,350)-(436,371): text "%.0f bar"; shows P307.Bar; alarm colour if P307.Alarm.Adver; runs INTERN ASSIGN INPUTS.PresSelCalStbd[9]:=(FALSE)
rectangle at (355,430)-(436,451): text "%.1f %%"; shows LS307.Pos; alarm colour if LS307.Alarm.Adver; runs INTERN ASSIGN INPUTS.PresSelCalStbd[9]:=(FALSE)
rectangle at (355,390)-(436,411): text "%.0f Kg"; shows L307.Kg; runs INTERN ASSIGN INPUTS.PresSelCalStbd[9]:=(FALSE)
rectangle at (0,0)-(1,1): text "{ExtendedElement},Visu\ElementDLL.ete,1,@Bargraph,86,21,3,0,0,LS307.Pos,,%,25,50,0,100,0,0,0,0,0,0,0,-13,16,700,Arial,0,255,0,255,0,0,0,0,0,0,0,0,0,,0,"
rectangle at (0,0)-(44,21): alarm colour if (LS307.Pos) < 0; right ((LS307.Pos * 1.0) - 50)  * 0.86
ellipse at (360,165)-(431,236): alarm colour if MAIN.fbSE307.OUT_CylIn
ellipse at (360,245)-(431,316): alarm colour if MAIN.fbSE307.OUT_CylOut
ellipse at (370,175)-(421,226): text "IN"; alarm colour if MAIN.fbSE307.IN_Hmi_CylIn; taps MAIN.fbSE307.IN_Hmi_CylIn
ellipse at (370,255)-(421,306): text "OUT"; alarm colour if MAIN.fbSE307.IN_Hmi_CylOut; taps MAIN.fbSE307.IN_Hmi_CylOut
rectangle at (370,60)-(421,81): text "J4"
rectangle at (355,335)-(426,351): text "P307"
rectangle at (355,375)-(426,391): text "L307"
rectangle at (355,415)-(426,431): text "LS307"
ellipse at (355,485)-(396,506): text "IN"; alarm colour if MAIN.fbSE307.LS_In
ellipse at (395,485)-(436,506): text "OUT"; alarm colour if MAIN.fbSE307.LS_Out
rounded rectangle at (40,100)-(111,136): text "ENABLE"; alarm colour if MAIN.aHP_Enable[1]; toggles MAIN.aHP_Enable[1]
rounded rectangle at (140,100)-(211,136): text "ENABLE"; alarm colour if MAIN.aHP_Enable[2]; toggles MAIN.aHP_Enable[2]
rounded rectangle at (250,100)-(321,136): text "ENABLE"; alarm colour if MAIN.aHP_Enable[3]; toggles MAIN.aHP_Enable[3]
rounded rectangle at (360,100)-(431,136): text "ENABLE"; alarm colour if MAIN.aHP_Enable[4]; toggles MAIN.aHP_Enable[4]
rounded rectangle at (905,450)-(1016,491): text "NEXT"; opens VISU_1_CYLINDERS2
rounded rectangle at (905,395)-(1016,436): text "CONFIG: / CYLINDERS1"; opens VISU_CFG_CYLINDERS1
rectangle at (465,350)-(546,371): text "%.0f bar"; shows P309.Bar; alarm colour if P309.Alarm.Adver; runs INTERN ASSIGN INPUTS.PresSelCalStbd[9]:=(FALSE)
rectangle at (465,390)-(546,411): text "%.0f Kg"; shows L309.Kg; runs INTERN ASSIGN INPUTS.PresSelCalStbd[9]:=(FALSE)
ellipse at (470,165)-(541,236): alarm colour if MAIN.fbSE309.OUT_CylIn
ellipse at (470,245)-(541,316): alarm colour if MAIN.fbSE309.OUT_CylOut
ellipse at (480,175)-(531,226): text "IN"; alarm colour if MAIN.fbSE309.IN_Hmi_CylIn; taps MAIN.fbSE309.IN_Hmi_CylIn
ellipse at (480,255)-(531,306): text "OUT"; alarm colour if MAIN.fbSE309.IN_Hmi_CylOut; taps MAIN.fbSE309.IN_Hmi_CylOut
rectangle at (470,60)-(541,81): text "FORESTAY"
rectangle at (465,335)-(536,351): text "P309"
rectangle at (465,375)-(536,391): text "L309"
rounded rectangle at (470,100)-(541,136): text "ENABLE"; alarm colour if MAIN.aHP_Enable[5]; toggles MAIN.aHP_Enable[5]
rectangle at (575,350)-(656,371): text "%.0f bar"; shows P311.Bar; alarm colour if P311.Alarm.Adver; runs INTERN ASSIGN INPUTS.PresSelCalStbd[9]:=(FALSE)
rectangle at (575,430)-(656,451): text "%.1f %%"; shows LS311.Pos; alarm colour if LS311.Alarm.Adver; runs INTERN ASSIGN INPUTS.PresSelCalStbd[9]:=(FALSE)
rectangle at (575,390)-(656,411): text "%.0f Kg"; shows L311.Kg; runs INTERN ASSIGN INPUTS.PresSelCalStbd[9]:=(FALSE)
rectangle at (0,0)-(1,1): text "{ExtendedElement},Visu\ElementDLL.ete,1,@Bargraph,86,21,3,0,0,LS311.Pos,,%,25,50,0,100,0,0,0,0,0,0,0,-13,16,700,Arial,0,255,0,255,0,0,0,0,0,0,0,0,0,,0,"
rectangle at (0,0)-(44,21): alarm colour if (LS311.Pos) < 0; right ((LS311.Pos * 1.0) - 50)  * 0.86
ellipse at (580,165)-(651,236): alarm colour if MAIN.fbSE311.OUT_CylIn
ellipse at (580,245)-(651,316): alarm colour if MAIN.fbSE311.OUT_CylOut
ellipse at (590,175)-(641,226): text "IN"; alarm colour if MAIN.fbSE311.IN_Hmi_CylIn; taps MAIN.fbSE311.IN_Hmi_CylIn
ellipse at (590,255)-(641,306): text "OUT"; alarm colour if MAIN.fbSE311.IN_Hmi_CylOut; taps MAIN.fbSE311.IN_Hmi_CylOut
rectangle at (575,335)-(646,351): text "P311"
rectangle at (575,375)-(646,391): text "L311"
rectangle at (575,415)-(646,431): text "LS311"
ellipse at (575,485)-(616,506): text "IN"; alarm colour if MAIN.fbSE311.LS_In
ellipse at (615,485)-(656,506): text "OUT"; alarm colour if MAIN.fbSE311.LS_Out
rounded rectangle at (580,100)-(651,136): text "ENABLE"; alarm colour if MAIN.aHP_Enable[6]; toggles MAIN.aHP_Enable[6]
rectangle at (590,60)-(641,81): text "J2"
rectangle at (690,55)-(761,86): text "SPARE1"
rectangle at (790,55)-(861,86): text "SPARE2"
rounded rectangle at (740,100)-(811,136): text "ENABLE"; alarm colour if MAIN.aHP_Enable[17]; toggles MAIN.aHP_Enable[17]
rectangle at (785,350)-(866,371): text "%.0f bar"; shows P903.Bar; alarm colour if P903.Alarm.Adver; runs INTERN ASSIGN INPUTS.PresSelCalStbd[9]:=(FALSE)
rectangle at (785,430)-(866,451): text "%.1f %%"; shows LS903.Pos; alarm colour if LS903.Alarm.Adver; runs INTERN ASSIGN INPUTS.PresSelCalStbd[9]:=(FALSE)
rectangle at (785,390)-(866,411): text "%.0f Kg"; shows L903.Kg; runs INTERN ASSIGN INPUTS.PresSelCalStbd[9]:=(FALSE)
rectangle at (0,0)-(1,1): text "{ExtendedElement},Visu\ElementDLL.ete,1,@Bargraph,86,21,3,0,0,LS903.Pos,,%,25,50,0,100,0,0,0,0,0,0,0,-13,16,700,Arial,0,255,0,255,0,0,0,0,0,0,0,0,0,,0,"
rectangle at (0,0)-(44,21): alarm colour if (LS903.Pos) < 0; right ((LS903.Pos * 1.0) - 50)  * 0.86
ellipse at (790,165)-(861,236): alarm colour if MAIN.fbBSY.OUT_S_In
ellipse at (790,245)-(861,316): alarm colour if MAIN.fbBSY.OUT_S_Out
ellipse at (800,175)-(851,226): text "IN"; alarm colour if MAIN.fbBSY.IN_Hmi_S_In; taps MAIN.fbBSY.IN_Hmi_S_In
ellipse at (800,255)-(851,306): text "OUT"; alarm colour if MAIN.fbBSY.IN_Hmi_S_Out; taps MAIN.fbBSY.IN_Hmi_S_Out
rectangle at (785,335)-(856,351): text "P903"
rectangle at (785,375)-(856,391): text "L903"
rectangle at (785,415)-(856,431): text "LS903"
ellipse at (785,485)-(826,506): text "IN"; alarm colour if MAIN.fbBSY.LS_S_In
ellipse at (825,485)-(866,506): text "OUT"; alarm colour if MAIN.fbBSY.LS_S_Out
rounded rectangle at (905,340)-(1016,381): text "CALIB: / CYLINDERS1"; opens VISU_CAL_CYLINDERS1
rectangle at (150,55)-(201,86): text "A3 / TACK"
rectangle at (50,55)-(101,86): text "FRO / TACK"
rectangle at (465,430)-(546,451): text "%.1f %%"; shows LS309.Pos; alarm colour if LS309.Alarm.Adver; runs INTERN ASSIGN INPUTS.PresSelCalStbd[9]:=(FALSE)
rectangle at (0,0)-(1,1): text "{ExtendedElement},Visu\ElementDLL.ete,1,@Bargraph,86,21,3,0,0,LS309.Pos,,%,25,50,0,100,0,0,0,0,0,0,0,-13,16,700,Arial,0,255,0,255,0,0,0,0,0,0,0,0,0,,0,"
rectangle at (0,0)-(44,21): alarm colour if (LS309.Pos) < 0; right ((LS309.Pos * 1.0) - 50)  * 0.86
rectangle at (465,415)-(536,431): text "LS309"
ellipse at (465,485)-(506,506): text "IN"; alarm colour if MAIN.fbSE309.LS_In
ellipse at (505,485)-(546,506): text "OUT"; alarm colour if MAIN.fbSE309.LS_Out
rounded rectangle at (905,55)-(1016,96): text "CLEAR"; alarm colour if ALARMS.Clear; taps ALARMS.Clear
rounded rectangle at (905,230)-(1016,271): text "MAST SETUP"; opens VISU_MAST_SETUP
27 more shapes without text or variables
*)

(* Visualisation VISU_1_CYLINDERS2
rectangle at (20,550)-(331,601): text "%s"; shows INPUTS.sVisuTime
rounded rectangle at (905,505)-(1016,546): text "RETURN"; opens VISU_0_MAIN
rectangle at (20,0)-(331,51): text "CYLINDERS 2"
rounded rectangle at (905,450)-(1016,491): text "BACK"; opens VISU_1_CYLINDERS1
rounded rectangle at (905,395)-(1016,436): text "CONFIG: / CYLINDERS2"; opens VISU_CFG_CYLINDERS2
rounded rectangle at (905,340)-(1016,381): text "CALIB: / CYLINDERS2"; opens VISU_CAL_CYLINDERS2
rectangle at (35,350)-(116,371): text "%.0f bar"; shows P501.Bar; alarm colour if P501.Alarm.Adver; runs INTERN ASSIGN INPUTS.PresSelCalStbd[9]:=(FALSE)
rectangle at (35,430)-(116,451): text "%.0f Kg"; shows L501_7; runs INTERN ASSIGN INPUTS.PresSelCalStbd[9]:=(FALSE)
ellipse at (40,165)-(111,236): alarm colour if MAIN.fbSE501.OUT_CylIn
ellipse at (40,245)-(111,316): alarm colour if MAIN.fbSE501.OUT_CylOut
ellipse at (50,175)-(101,226): text "IN"; alarm colour if MAIN.fbSE501.IN_Hmi_CylIn; taps MAIN.fbSE501.IN_Hmi_CylIn
ellipse at (50,255)-(101,306): text "OUT"; alarm colour if MAIN.fbSE501.IN_Hmi_CylOut; taps MAIN.fbSE501.IN_Hmi_CylOut
rectangle at (35,335)-(106,351): text "P501"
rectangle at (35,415)-(106,431): text "L501-L507"
rectangle at (135,350)-(216,371): text "%.0f bar"; shows P503.Bar; alarm colour if P503.Alarm.Adver; runs INTERN ASSIGN INPUTS.PresSelCalStbd[9]:=(FALSE)
rectangle at (135,390)-(216,411): text "%.0f Kg"; shows L503.Kg; runs INTERN ASSIGN INPUTS.PresSelCalStbd[9]:=(FALSE)
ellipse at (140,165)-(211,236): alarm colour if MAIN.fbSE503.OUT_CylIn
ellipse at (140,245)-(211,316): alarm colour if MAIN.fbSE503.OUT_CylOut
ellipse at (150,175)-(201,226): text "IN"; alarm colour if MAIN.fbSE503.IN_Hmi_CylIn; taps MAIN.fbSE503.IN_Hmi_CylIn
ellipse at (150,255)-(201,306): text "OUT"; alarm colour if MAIN.fbSE503.IN_Hmi_CylOut; taps MAIN.fbSE503.IN_Hmi_CylOut
rectangle at (135,335)-(206,351): text "P503"
rectangle at (135,375)-(206,391): text "L503"
rectangle at (245,350)-(326,371): text "%.0f bar"; shows P505.Bar; alarm colour if P505.Alarm.Adver; runs INTERN ASSIGN INPUTS.PresSelCalStbd[9]:=(FALSE)
rectangle at (245,390)-(326,411): text "%.0f Kg"; shows L505.Kg; runs INTERN ASSIGN INPUTS.PresSelCalStbd[9]:=(FALSE)
ellipse at (250,165)-(321,236): alarm colour if MAIN.fbSE505.OUT_CylIn
ellipse at (250,245)-(321,316): alarm colour if MAIN.fbSE505.OUT_CylOut
ellipse at (260,175)-(311,226): text "IN"; alarm colour if MAIN.fbSE505.IN_Hmi_CylIn; taps MAIN.fbSE505.IN_Hmi_CylIn
ellipse at (260,255)-(311,306): text "OUT"; alarm colour if MAIN.fbSE505.IN_Hmi_CylOut; taps MAIN.fbSE505.IN_Hmi_CylOut
rectangle at (260,60)-(311,81): text "SPARE3"
rectangle at (245,335)-(316,351): text "P505"
rectangle at (245,375)-(316,391): text "L505"
rounded rectangle at (40,100)-(111,136): text "ENABLE"; alarm colour if MAIN.aHP_Enable[7]; toggles MAIN.aHP_Enable[7]
rounded rectangle at (140,100)-(211,136): text "ENABLE"; alarm colour if MAIN.aHP_Enable[8]; toggles MAIN.aHP_Enable[8]
rounded rectangle at (250,100)-(321,136): text "ENABLE"; alarm colour if MAIN.aHP_Enable[9]; toggles MAIN.aHP_Enable[9]
rectangle at (50,55)-(101,86): text "JIB / IN/OUT"
rectangle at (150,55)-(201,86): text "JIB / UP/DW"
rectangle at (355,350)-(436,371): text "%.0f bar"; shows P701.Bar; alarm colour if P701.Alarm.Adver; runs INTERN ASSIGN INPUTS.PresSelCalStbd[9]:=(FALSE)
rectangle at (685,430)-(766,451): text "%.1f %%"; shows LS707.Pos; alarm colour if LS707.Alarm.Adver; runs INTERN ASSIGN INPUTS.PresSelCalStbd[9]:=(FALSE)
rectangle at (355,390)-(436,411): text "%.0f Kg"; shows L701.Kg; runs INTERN ASSIGN INPUTS.PresSelCalStbd[9]:=(FALSE)
rectangle at (0,0)-(1,1): text "{ExtendedElement},Visu\ElementDLL.ete,1,@Bargraph,86,21,3,0,0,LS707.Pos,,%,25,50,0,100,0,0,0,0,0,0,0,-13,16,700,Arial,0,255,0,255,0,0,0,0,0,0,0,0,0,,0,"
rectangle at (0,0)-(44,21): alarm colour if (LS707.Pos) < 0; right ((LS707.Pos * 1.0) - 50)  * 0.86
ellipse at (360,165)-(431,236): alarm colour if MAIN.fbSE701.OUT_CylIn
ellipse at (360,245)-(431,316): alarm colour if MAIN.fbSE701.OUT_CylOut
ellipse at (370,175)-(421,226): text "IN"; alarm colour if MAIN.fbSE701.IN_Hmi_CylIn; taps MAIN.fbSE701.IN_Hmi_CylIn
ellipse at (370,255)-(421,306): text "OUT"; alarm colour if MAIN.fbSE701.IN_Hmi_CylOut; taps MAIN.fbSE701.IN_Hmi_CylOut
rectangle at (355,335)-(426,351): text "P701"
rectangle at (355,375)-(426,391): text "L701"
rectangle at (685,415)-(756,431): text "LS707"
ellipse at (685,485)-(726,506): text "IN"; alarm colour if MAIN.fbSE707.LS_In
ellipse at (725,485)-(766,506): text "OUT"; alarm colour if MAIN.fbSE707.LS_Out
rectangle at (465,350)-(546,371): text "%.0f bar"; shows P703.Bar; alarm colour if P703.Alarm.Adver; runs INTERN ASSIGN INPUTS.PresSelCalStbd[9]:=(FALSE)
rectangle at (785,430)-(866,451): text "%.1f %%"; shows LS709.Pos; alarm colour if LS709.Alarm.Adver; runs INTERN ASSIGN INPUTS.PresSelCalStbd[9]:=(FALSE)
rectangle at (465,390)-(546,411): text "%.0f Kg"; shows L703.Kg; runs INTERN ASSIGN INPUTS.PresSelCalStbd[9]:=(FALSE)
rectangle at (0,0)-(1,1): text "{ExtendedElement},Visu\ElementDLL.ete,1,@Bargraph,86,21,3,0,0,LS709.Pos,,%,25,50,0,100,0,0,0,0,0,0,0,-13,16,700,Arial,0,255,0,255,0,0,0,0,0,0,0,0,0,,0,"
rectangle at (0,0)-(44,21): alarm colour if (LS709.Pos) < 0; right ((LS709.Pos * 1.0) - 50)  * 0.86
ellipse at (470,165)-(541,236): alarm colour if MAIN.fbSE703.OUT_CylIn
ellipse at (470,245)-(541,316): alarm colour if MAIN.fbSE703.OUT_CylOut
ellipse at (480,175)-(531,226): text "IN"; alarm colour if MAIN.fbSE703.IN_Hmi_CylIn; taps MAIN.fbSE703.IN_Hmi_CylIn
ellipse at (480,255)-(531,306): text "OUT"; alarm colour if MAIN.fbSE703.IN_Hmi_CylOut; taps MAIN.fbSE703.IN_Hmi_CylOut
rectangle at (465,335)-(536,351): text "P703"
rectangle at (465,375)-(536,391): text "L703"
rectangle at (785,415)-(856,431): text "LS709"
ellipse at (785,485)-(826,506): text "IN"; alarm colour if MAIN.fbSE709.LS_In
ellipse at (825,485)-(866,506): text "OUT"; alarm colour if MAIN.fbSE709.LS_Out
rectangle at (575,350)-(656,371): text "%.0f bar"; shows P705.Bar; alarm colour if P705.Alarm.Adver; runs INTERN ASSIGN INPUTS.PresSelCalStbd[9]:=(FALSE)
rectangle at (575,390)-(656,411): text "%.0f Kg"; shows L705.Kg; runs INTERN ASSIGN INPUTS.PresSelCalStbd[9]:=(FALSE)
ellipse at (580,165)-(651,236): alarm colour if MAIN.fbSE705.OUT_CylIn
ellipse at (580,245)-(651,316): alarm colour if MAIN.fbSE705.OUT_CylOut
ellipse at (590,175)-(641,226): text "IN"; alarm colour if MAIN.fbSE705.IN_Hmi_CylIn; taps MAIN.fbSE705.IN_Hmi_CylIn
ellipse at (590,255)-(641,306): text "OUT"; alarm colour if MAIN.fbSE705.IN_Hmi_CylOut; taps MAIN.fbSE705.IN_Hmi_CylOut
rectangle at (575,335)-(646,351): text "P705"
rectangle at (575,375)-(646,391): text "L705"
rectangle at (685,350)-(766,371): text "%.0f bar"; shows P707.Bar; alarm colour if P707.Alarm.Adver; runs INTERN ASSIGN INPUTS.PresSelCalStbd[9]:=(FALSE)
rectangle at (685,390)-(766,411): text "%.0f Kg"; shows L707.Kg; runs INTERN ASSIGN INPUTS.PresSelCalStbd[9]:=(FALSE)
ellipse at (690,165)-(761,236): alarm colour if MAIN.fbSE707.OUT_CylIn
ellipse at (690,245)-(761,316): alarm colour if MAIN.fbSE707.OUT_CylOut
ellipse at (700,175)-(751,226): text "IN"; alarm colour if MAIN.fbSE707.IN_Hmi_CylIn; taps MAIN.fbSE707.IN_Hmi_CylIn
ellipse at (700,255)-(751,306): text "OUT"; alarm colour if MAIN.fbSE707.IN_Hmi_CylOut; taps MAIN.fbSE707.IN_Hmi_CylOut
rectangle at (685,335)-(756,351): text "P707"
rectangle at (685,375)-(756,391): text "L707"
rounded rectangle at (360,100)-(431,136): text "ENABLE"; alarm colour if MAIN.aHP_Enable[12]; toggles MAIN.aHP_Enable[12]
rounded rectangle at (470,100)-(541,136): text "ENABLE"; alarm colour if MAIN.aHP_Enable[13]; toggles MAIN.aHP_Enable[13]
rounded rectangle at (580,100)-(651,136): text "ENABLE"; alarm colour if MAIN.aHP_Enable[14]; toggles MAIN.aHP_Enable[14]
rounded rectangle at (690,100)-(761,136): text "ENABLE"; alarm colour if MAIN.aHP_Enable[15]; toggles MAIN.aHP_Enable[15]
rectangle at (785,350)-(866,371): text "%.0f bar"; shows P709.Bar; alarm colour if P709.Alarm.Adver; runs INTERN ASSIGN INPUTS.PresSelCalStbd[9]:=(FALSE)
rectangle at (785,390)-(866,411): text "%.0f Kg"; shows L709.Kg; runs INTERN ASSIGN INPUTS.PresSelCalStbd[9]:=(FALSE)
ellipse at (790,165)-(861,236): alarm colour if MAIN.fbSE709.OUT_CylIn
ellipse at (790,245)-(861,316): alarm colour if MAIN.fbSE709.OUT_CylOut
ellipse at (800,175)-(851,226): text "IN"; alarm colour if MAIN.fbSE709.IN_Hmi_CylIn; taps MAIN.fbSE709.IN_Hmi_CylIn
ellipse at (800,255)-(851,306): text "OUT"; alarm colour if MAIN.fbSE709.IN_Hmi_CylOut; taps MAIN.fbSE709.IN_Hmi_CylOut
rectangle at (785,335)-(856,351): text "P709"
rectangle at (785,375)-(856,391): text "L709"
rounded rectangle at (790,100)-(861,136): text "ENABLE"; alarm colour if MAIN.aHP_Enable[16]; toggles MAIN.aHP_Enable[16]
rectangle at (685,55)-(756,86): text "BOTTOM / DEFLECTOR"
rectangle at (790,55)-(861,86): text "TOP / DEFLECTOR"
rectangle at (360,55)-(431,86): text "INNER / STAYSAIL"
rectangle at (470,55)-(541,86): text "MAIN / OUTHAUL"
rectangle at (580,55)-(651,86): text "MAIN / CUNN"
rectangle at (35,390)-(116,411): text "%.0f bar"; shows P507.Bar; alarm colour if P507.Alarm.Adver; runs INTERN ASSIGN INPUTS.PresSelCalStbd[9]:=(FALSE)
rectangle at (35,375)-(106,391): text "P507"
rounded rectangle at (905,55)-(1016,96): text "CLEAR"; alarm colour if ALARMS.Clear; taps ALARMS.Clear
21 more shapes without text or variables
*)

